# B&R Automation Studio project mappFramework (part 2)

#### HelperMacro.h
```c
/*
* Author: 		B+R
* Contents of this file are modified and extended
*/

/*
 * COPYRIGHT AND PERMISSION NOTICE
 *
 * Copyright (c) 2003 Embedded Unit Project
 *
 * All rights reserved.
 *
 * Permission is hereby granted, free of charge, to any person obtaining
 * a copy of this software and associated documentation files (the
 * "Software"), to deal in the Software without restriction, including
 * without limitation the rights to use, copy, modify, merge, publish,
 * distribute, and/or sell copies of the Software, and to permit persons
 * to whom the Software is furnished to do so, provided that the above
 * copyright notice(s) and this permission notice appear in all copies
 * of the Software and that both the above copyright notice(s) and this
 * permission notice appear in supporting documentation.
 *
 * THE SOFTWARE IS PROVIDED "AS IS", WITHOUT WARRANTY OF ANY KIND,
 * EXPRESS OR IMPLIED, INCLUDING BUT NOT LIMITED TO THE WARRANTIES OF
 * MERCHANTABILITY, FITNESS FOR A PARTICULAR PURPOSE AND NONINFRINGEMENT
 * OF THIRD PARTY RIGHTS. IN NO EVENT SHALL THE COPYRIGHT HOLDER OR
 * HOLDERS INCLUDED IN THIS NOTICE BE LIABLE FOR ANY CLAIM, OR ANY
 * SPECIAL INDIRECT OR CONSEQUENTIAL DAMAGES, OR ANY DAMAGES WHATSOEVER
 * RESULTING FROM LOSS OF USE, DATA OR PROFITS, WHETHER IN AN ACTION OF
 * CONTRACT, NEGLIGENCE OR OTHER TORTIOUS ACTION, ARISING OUT OF OR IN
 * CONNECTION WITH THE USE OR PERFORMANCE OF THIS SOFTWARE.
 *
 * Except as contained in this notice, the name of a copyright holder
 * shall not be used in advertising or otherwise to promote the sale,
 * use or other dealings in this Software without prior written
 * authorization of the copyright holder.
 *
 * $Id: HelperMacro.h,v 1.3 2004/02/10 16:19:29 arms22 Exp $
 */

#ifndef	__HELPERMACRO_H__
#define	__HELPERMACRO_H__

/* Defines the order of test cases */
#define UNITTEST_FIXTURES(fixtures) \
	static const TestFixture	fixtures[] =

/* Standard UnitTest caller without any setup / teardown methods*/
#define UNITTEST_CALLER_TEST(caller,name,fixtures) \
	UNITTEST_CALLER_COMPLETE_EXPLICIT(caller,name,0,0,fixtures,0,0, 0)

/* Standard UnitTest caller with macro setup / teardown for tests*/
#define UNITTEST_CALLER_BASIC(caller,name,fixtures) \
	UNITTEST_CALLER_COMPLETE_EXPLICIT(caller,name,setupTest,teardownTest,fixtures,0,0, 0)

/* UnitTest caller with macro setup / teardown for tests and test set */
#define UNITTEST_CALLER_SET(caller,name,fixtures) \
	UNITTEST_CALLER_COMPLETE_EXPLICIT(caller,name,setupTest,teardownTest,fixtures, setupSet, teardownSet, 0)

/* UnitTest caller with macro setup / teardown for tests and test set and cylic*/
#define UNITTEST_CALLER_COMPLETE(caller,name,fixtures) \
	UNITTEST_CALLER_COMPLETE_EXPLICIT(caller,name,setupTest,teardownTest,fixtures, setupSet, teardownSet, cyclicSetCaller)

/* UnitTest caller with explicit setup / teardown for suite */
#define UNITTEST_CALLER_SET_EXPLICIT(caller,name,sup,tdw,fixtures, setupSuite, teardownSuite) \
	UNITTEST_CALLER_COMPLETE_EXPLICIT(caller,name,sup,tdw,fixtures, setupSuite, teardownSuite, 0)

#ifdef  __cplusplus
/* UnitTest caller with explicit setup / teardown for suite and cylic */
#define UNITTEST_CALLER_COMPLETE_EXPLICIT(caller,name,sup,tdw,fixtures, setupSuite, teardownSuite, cyclicCaller) \
	UNITTEST_TESTSET_DECLARATION caller = new_TestCaller(name,sup,tdw,sizeof(fixtures)/sizeof(fixtures[0]),(TestFixture*)fixtures, setupSuite, teardownSuite, cyclicCaller)

#else

/* UnitTest caller with explicit setup / teardown for suite and cylic */
#define UNITTEST_CALLER_COMPLETE_EXPLICIT(caller,name,sup,tdw,fixtures, setupSuite, teardownSuite, cyclicCaller) \
	 const TestCaller caller = new_TestCaller(name,sup,tdw,sizeof(fixtures)/sizeof(fixtures[0]),(TestFixture*)fixtures, setupSuite, teardownSuite, cyclicCaller)

#endif

#define UNITTEST_CALLER_SKIPPED(caller,name,sup,tdw,fixtures, setupSuite, teardownSuite, cyclicCaller) \
 const TestCaller caller = skipTestCaller(name,sup,tdw,sizeof(fixtures)/sizeof(fixtures[0]),(TestFixture*)fixtures, setupSuite, teardownSuite, cyclicCaller)

/* --------------------------------------*/

/* --------------------------------------*/

typedef struct TestSetActive
{
	BOOL			active;
	TestCallerRef 	set;
} TestSetActive;

typedef struct TestSetList
{
	UINT 			nrOfTestSets;
	UINT 			currentTestSet;
	TestSetActive 	*list;
} TestSetList;

/* Defines the order of test sets.
Should look like this
UNITTEST_TESTSET_FIXTURES(fixtures)
{
	new_TestSet(testSet_1),
	new_TestSet(testSet_2),
	new_TestSet(testSet_3)
}*/
#define UNITTEST_TESTSET_FIXTURES(fixtures) \
	static TestSetActive	fixtures[] =

/* Adds a test set with description to the fixture of test sets.
See UNITTEST_TESTSET_FIXTURES() */
#define new_TestSet(testcaller)\
	{\
		1,\
		(TestCallerRef)&testcaller,\
	}

/* Adds a test set with description to the fixture of test sets.
See UNITTEST_TESTSET_FIXTURES() */
#define skipTestSet(testcaller)\
	{\
		1,\
		(TestCallerRef)&testcaller,\
	}

/* Adds a test set with description to the fixture of test sets.
See UNITTEST_TESTSET_FIXTURES() */
#define disabledTestSet(testcaller)\
	{\
		0,\
		(TestCallerRef)&testcaller,\
	}

/* Defines the test set list handling structure*/
#define UNTITTEST_TESTSET_HANDLER() \
TestSetList setList = {\
	sizeof(utTestSets) / sizeof(TestSetActive), \
	0, \
	(TestSetActive*)&utTestSets\
	}

#endif/*__HELPERMACRO_H__*/
```

#### utRunner.h
```c
/********************************************************************
 * COPYRIGHT B+R
 ********************************************************************
 * Library: utRunner
 * File: utRunner.h
 * Author: B+R
 *******************************************************************/

#ifndef	__UT_RUNNER_H__
#define	__UT_RUNNER_H__

#include <bur/plctypes.h>

#include "UnitTest.h"
#include "UtMgr.h"
#include "include/TestCaller.h"

#ifdef __cplusplus
extern "C"
{
#endif

void utInit(UtMgrTestSuite_typ *TestSuiteRef);
void utCyclic(UtMgrTestSuite_typ *TestSuiteRef);
void utExit(UtMgrTestSuite_typ *TestSuiteRef);

#ifdef __cplusplus
};
#endif

#endif/*__UT_RUNNER_H__*/
```

#### Test.h
```c
/*
* Author: 		B+R
* Contents of this file are modified and extended
*/

/*
 * COPYRIGHT AND PERMISSION NOTICE
 *
 * Copyright (c) 2003 Embedded Unit Project
 *
 * All rights reserved.
 *
 * Permission is hereby granted, free of charge, to any person obtaining
 * a copy of this software and associated documentation files (the
 * "Software"), to deal in the Software without restriction, including
 * without limitation the rights to use, copy, modify, merge, publish,
 * distribute, and/or sell copies of the Software, and to permit persons
 * to whom the Software is furnished to do so, provided that the above
 * copyright notice(s) and this permission notice appear in all copies
 * of the Software and that both the above copyright notice(s) and this
 * permission notice appear in supporting documentation.
 *
 * THE SOFTWARE IS PROVIDED "AS IS", WITHOUT WARRANTY OF ANY KIND,
 * EXPRESS OR IMPLIED, INCLUDING BUT NOT LIMITED TO THE WARRANTIES OF
 * MERCHANTABILITY, FITNESS FOR A PARTICULAR PURPOSE AND NONINFRINGEMENT
 * OF THIRD PARTY RIGHTS. IN NO EVENT SHALL THE COPYRIGHT HOLDER OR
 * HOLDERS INCLUDED IN THIS NOTICE BE LIABLE FOR ANY CLAIM, OR ANY
 * SPECIAL INDIRECT OR CONSEQUENTIAL DAMAGES, OR ANY DAMAGES WHATSOEVER
 * RESULTING FROM LOSS OF USE, DATA OR PROFITS, WHETHER IN AN ACTION OF
 * CONTRACT, NEGLIGENCE OR OTHER TORTIOUS ACTION, ARISING OUT OF OR IN
 * CONNECTION WITH THE USE OR PERFORMANCE OF THIS SOFTWARE.
 *
 * Except as contained in this notice, the name of a copyright holder
 * shall not be used in advertising or otherwise to promote the sale,
 * use or other dealings in this Software without prior written
 * authorization of the copyright holder.
 *
 * $Id: Test.h,v 1.4 2004/02/10 16:19:29 arms22 Exp $
 */
#ifndef	__TEST_H__
#define	__TEST_H__

typedef struct __TestResult		TestResult;
typedef struct __TestResult	*TestResultRef;/*downward compatible*/

typedef struct __TestImplement	TestImplement;
typedef struct __TestImplement	*TestImplementRef;/*downward compatible*/

typedef enum testStatusEnum
{
    ut_BUSY = 0,
    ut_DONE = 1,
    ut_ABORT = 2
} testStatusEnum;

typedef char* 			(*TestNameFunction)(void *);

typedef testStatusEnum	(*TestRunFunction)(void *, TestResult *);
typedef int				(*TestCountTestCasesFunction)(void *);

typedef enum testStateEnum
{
    stateStart, 	/* print something */
    stateSetup,
    stateRun,
    stateTearDown,
    stateEnd,		/* print something */
    stateDefault, 	/* last state*/
} testStateEnum;

struct __TestImplement
{
	TestNameFunction 			name;
	TestRunFunction 			run;
	TestCountTestCasesFunction countTestCases;
};

typedef struct __Test	Test;
typedef struct __Test	*TestRef;/*downward compatible*/

struct __Test
{
	TestImplement *isa;
};

#define Test_name(s)			((Test*)s)->isa->name(s)
#define Test_run(s,r)			((Test*)s)->isa->run(s,r)
#define Test_countTestCases(s)	((Test*)s)->isa->countTestCases(s)

#endif/*__TEST_H__*/
```

#### TestListener.h
```c
/*
* Author: 		B+R
* Contents of this file are modified and extended
*/

/*
 * COPYRIGHT AND PERMISSION NOTICE
 *
 * Copyright (c) 2003 Embedded Unit Project
 *
 * All rights reserved.
 *
 * Permission is hereby granted, free of charge, to any person obtaining
 * a copy of this software and associated documentation files (the
 * "Software"), to deal in the Software without restriction, including
 * without limitation the rights to use, copy, modify, merge, publish,
 * distribute, and/or sell copies of the Software, and to permit persons
 * to whom the Software is furnished to do so, provided that the above
 * copyright notice(s) and this permission notice appear in all copies
 * of the Software and that both the above copyright notice(s) and this
 * permission notice appear in supporting documentation.
 *
 * THE SOFTWARE IS PROVIDED "AS IS", WITHOUT WARRANTY OF ANY KIND,
 * EXPRESS OR IMPLIED, INCLUDING BUT NOT LIMITED TO THE WARRANTIES OF
 * MERCHANTABILITY, FITNESS FOR A PARTICULAR PURPOSE AND NONINFRINGEMENT
 * OF THIRD PARTY RIGHTS. IN NO EVENT SHALL THE COPYRIGHT HOLDER OR
 * HOLDERS INCLUDED IN THIS NOTICE BE LIABLE FOR ANY CLAIM, OR ANY
 * SPECIAL INDIRECT OR CONSEQUENTIAL DAMAGES, OR ANY DAMAGES WHATSOEVER
 * RESULTING FROM LOSS OF USE, DATA OR PROFITS, WHETHER IN AN ACTION OF
 * CONTRACT, NEGLIGENCE OR OTHER TORTIOUS ACTION, ARISING OUT OF OR IN
 * CONNECTION WITH THE USE OR PERFORMANCE OF THIS SOFTWARE.
 *
 * Except as contained in this notice, the name of a copyright holder
 * shall not be used in advertising or otherwise to promote the sale,
 * use or other dealings in this Software without prior written
 * authorization of the copyright holder.
 *
 * $Id: TestListener.h,v 1.4 2004/02/10 16:19:29 arms22 Exp $
 */
#ifndef	__TESTLISTENER_H__
#define	__TESTLISTENER_H__

typedef struct __TestListnerImplement	TestListnerImplement;
typedef struct __TestListnerImplement	*TestListnerImplementRef;/*downward compatible*/

typedef void(*TestListnerStartTestCallBack)(void *,void *);
typedef void(*TestListnerEndTestCallBack)(void *,void *);
typedef void(*TestListnerSkippedTestCallBack)(void *,void *);

typedef void(*TestListnerAddFailureCallBack)(void *,void *,const char *,unsigned long,const char *);

typedef void(*TestListnerAddPassedCallBack)(void *,void *,const char *,unsigned long,const char *);
typedef void(*TestListnerAddInfoCallBack)(void *,void *,const char *,unsigned long,const char *);
typedef void(*TestListnerAddAbortCallBack)(void *,void *,const char *,unsigned long,const char *);
typedef void(*TestListnerLogCallBack)(void *,void *,const char *,unsigned long,const char *, signed short);

struct __TestListnerImplement
{
	TestListnerStartTestCallBack 	startTest;
	TestListnerEndTestCallBack 		endTest;
	TestListnerSkippedTestCallBack 	skippedTest;
	TestListnerAddFailureCallBack 	addFailure;
	TestListnerAddPassedCallBack 	addPassed;
	TestListnerAddInfoCallBack 		addInfo;
	TestListnerAddAbortCallBack 	addAbort;
	TestListnerLogCallBack			doLog;
};

/*typedef struct __TestListner	TestListner;*/	/*->TestResult.h*/
/*typedef struct __TestListner*	TestListnerRef;*/	/*->TestResult.h*/

struct __TestListner
{
	TestListnerImplement *isa;
};

#define TestListner_startTest(s,t)			((TestListner*)s)->isa->startTest(s,t)
#define TestListner_endTest(s,t)			((TestListner*)s)->isa->endTest(s,t)
#define TestListner_skippedTest(s,t)			((TestListner*)s)->isa->skippedTest(s,t)

#define TestListner_addFailure(s,t,m,l,f)	((TestListner*)s)->isa->addFailure(s,t,m,l,f)
#define TestListner_addPassed(s,t,m,l,f)	((TestListner*)s)->isa->addPassed(s,t,m,l,f)
#define TestListner_addInfo(s,t,m,l,f)		((TestListner*)s)->isa->addInfo(s,t,m,l,f)
#define TestListner_addAbort(s,t,m,l,f)		((TestListner*)s)->isa->addAbort(s,t,m,l,f)
#define TestListener_doLog(s,t,m,l,f,e)		if(s)(((TestListner*)s)->isa->doLog(s,t,m,l,f,e))
#endif/*__TESTLISTENER_H__*/
```

#### TestResult.h
```c
/*
* Author: 		B+R
* Contents of this file are modified and extended
*/

/*
* COPYRIGHT AND PERMISSION NOTICE
*
* Copyright (c) 2003 Embedded Unit Project
*
* All rights reserved.
*
* Permission is hereby granted, free of charge, to any person obtaining
* a copy of this software and associated documentation files (the
* "Software"), to deal in the Software without restriction, including
* without limitation the rights to use, copy, modify, merge, publish,
* distribute, and/or sell copies of the Software, and to permit persons
* to whom the Software is furnished to do so, provided that the above
* copyright notice(s) and this permission notice appear in all copies
* of the Software and that both the above copyright notice(s) and this
* permission notice appear in supporting documentation.
*
* THE SOFTWARE IS PROVIDED "AS IS", WITHOUT WARRANTY OF ANY KIND,
* EXPRESS OR IMPLIED, INCLUDING BUT NOT LIMITED TO THE WARRANTIES OF
* MERCHANTABILITY, FITNESS FOR A PARTICULAR PURPOSE AND NONINFRINGEMENT
* OF THIRD PARTY RIGHTS. IN NO EVENT SHALL THE COPYRIGHT HOLDER OR
* HOLDERS INCLUDED IN THIS NOTICE BE LIABLE FOR ANY CLAIM, OR ANY
* SPECIAL INDIRECT OR CONSEQUENTIAL DAMAGES, OR ANY DAMAGES WHATSOEVER
* RESULTING FROM LOSS OF USE, DATA OR PROFITS, WHETHER IN AN ACTION OF
* CONTRACT, NEGLIGENCE OR OTHER TORTIOUS ACTION, ARISING OUT OF OR IN
* CONNECTION WITH THE USE OR PERFORMANCE OF THIS SOFTWARE.
*
* Except as contained in this notice, the name of a copyright holder
* shall not be used in advertising or otherwise to promote the sale,
* use or other dealings in this Software without prior written
* authorization of the copyright holder.
*
* $Id: TestResult.h,v 1.7 2004/02/10 16:19:29 arms22 Exp $
*/
#ifndef	__TESTRESULT_H__
#define	__TESTRESULT_H__

#ifdef	__cplusplus
extern "C" {
#endif

/*typedef struct __TestResult		TestResult;*//* -> Test.h*/
/*typedef struct __TestResult*		TestResultRef;*//* -> Test.h*/

typedef struct __TestListner	TestListner;
typedef struct __TestListner	*TestListnerRef;/*downward compatible*/

struct __TestResult
{
	unsigned short runCount;
	unsigned short failureCount;
	unsigned short passedCount;
	unsigned short infoCount;
	unsigned short summarizedCount;
	unsigned short abortCount;
	unsigned short skippedTestCount;
	unsigned short suceessedTestCount;
	TestListner *listener;
};

#define new_TestResult(listener)\
{\
	0,\
	0,\
	0,\
	0,\
	0,\
	0,\
	0,\
	0,\
	(TestListner*)listener\
}

void TestResult_init(TestResult *self,TestListner *listner);
void TestResult_startTest(TestResult *self,Test *test);
void TestResult_endTest(TestResult *self,Test *test);
void TestResult_skipTest(TestResult *self,Test *test);

void TestResult_addFailure(TestResult *self,Test *test,const char *msg,unsigned long line,const char *file);
void TestResult_addPassed(TestResult *self,Test *test,const char *msg,unsigned long line,const char *file);
void TestResult_addInfo(TestResult *self,Test *test,const char *msg,unsigned long line,const char *file);
void TestResult_addAbort(TestResult *self,Test *test,const char *msg,unsigned long line,const char *file);

#ifdef	__cplusplus
}
#endif

#endif/*__TESTRESULT_H__*/
```

### Package Logical/Infrastructure/TS_UnitTest/Samples/Tests_Program - Unit test sample

### Library Logical/Infrastructure/TS_UnitTest/Samples/Tests_Program/SPLMyCalc (IEC)
Depends on: Runtime

#### SPLMyCalc.st
```iecst
(********************************************************************
 * COPYRIGHT -- Bernecker + Rainer
 ********************************************************************
 * Library: SPLMyCalc
 * File: SPLMyCalc.st
 * Author: B+R
 ********************************************************************
 * Implementation of library SPLMyCalc
 *******************************************************************

// This can be used as a sample for  Test Driven Development (TDD)/ Test First Development
Steps (in a nutshell):
    o Define your API (FB, functions, ...)
		 this is already done for the FB MyCalc
	o Create a new test program (by using the template)
	o Write a test case (e.g. Addition) for this FB.
		The tests should describe the expected behavior.
	o Transfer the test program to the target and run the test in the test view
		The test case will fail
	o Implement this FB (Addition), build and transfer, then run the test again
		The test case will pass
	o Write next test (e.g. Subtraction).
	..
	o Write test for MIN / MAX (underflow/overflow)
   	o Run the tests to verify your implementation.

Note:
	The sample test program in SPL_MyCalcLib_C provides some test cases using this FB.

FUNCTION_BLOCK MyCalculator

	Status := ERR_NOTIMPLEMENTED;

END_FUNCTION_BLOCK
```

### Program Logical/Infrastructure/TS_UnitTest/Samples/Tests_Program/Tests_MyCalcLib_C/SPL_CalcTest (ANSIC) - Tests SPLMyCalc with library "UnitTest"

#### testSuite.c - Handling of program and test suite
```c
/********************************************************************
 * COPYRIGHT -- Bernecker + Rainer
 ********************************************************************
 * Program: SPL_CalcTest
 * Author: B+R
 ********************************************************************
 * Test registration and handshake
 ********************************************************************/

#include <bur/plctypes.h>

#ifdef _DEFAULT_INCLUDES
#include <AsDefault.h>
#endif

#include "UnitTest.h"

void _INIT initTestSuite(void)
{
	utInit(&Testsuite);
}

void _CYCLIC cyclicWithTest(void)
{
	utCyclic(&Testsuite);
}

void _EXIT exitTestSuite(void)
{
	utExit(&Testsuite);
}
```

#### testSet_MyCalcLib_Addition.c - Groups test cases for addition
```c
/********************************************************************
 * COPYRIGHT -- Bernecker + Rainer
 ********************************************************************
 * Program: SPL_CalcTest
 * Author: B+R
 ********************************************************************
 * Test set implementation
 ********************************************************************/

#include <bur/plctypes.h>

#ifdef _DEFAULT_INCLUDES
#include <AsDefault.h>
#endif

#include "UnitTest.h"

_TEST test_Add(void)
{
	/* initialize functionblock parameters */
	instMyCalc.CalcOperator = splMyCalcOPERATOR_ADD;
	instMyCalc.Param1   = 1;
	instMyCalc.Param2   = 2;
	/* call synchron functionblock */
	MyCalculator(&instMyCalc);

	/* check result */
	TEST_ASSERT_EQUAL_INT(3, instMyCalc.Result);
	TEST_ASSERT_EQUAL_INT(ERR_OK, instMyCalc.Status);

	/* test is done */
	TEST_DONE;
}

_TEST testResetOutputParam(void)
{

	/* Do any calculation with a result != 0  */
	instMyCalc.CalcOperator = splMyCalcOPERATOR_ADD;
	instMyCalc.Param1   = 1;
	instMyCalc.Param2   = 2;
	/* call synchron functionblock */
	MyCalculator(&instMyCalc);
	/* Please note: the result of the calculation isn't checked as this is not subject of this test case.	 */

	instMyCalc.CalcOperator = splMyCalcOPERATOR_RESET_OUTPUTS;
	/* call synchron functionblock */
	MyCalculator(&instMyCalc);

	/* check result */
	TEST_ASSERT_EQUAL_INT(0, instMyCalc.Result);
	TEST_ASSERT_EQUAL_INT(ERR_OK, instMyCalc.Status);

	/* test is done */
	TEST_DONE;

}

/* This test case shows an example of a test case that can be "false positive".
	As long as MyCalculator() is not implemented, this test passes.
	As long as instMyCalc.Result already is 0 when this test case will be called, it doesn't check wether the FB was called at all.
	--> There are several methods, to verify the FB was called and changed the variables that are used to prove functionality:
	Choose other parameter for an addition with negative values
	Before calling the FB set the output to any other value than the expected result. (e.g. By using _SETUP_TEST() and / or _TEARDOWN_TEST() )
	...

*/
_TEST test_Addition_negValue_badExampleParameter(void)
{
	/* initialize functionblock parameters */
	instMyCalc.CalcOperator = splMyCalcOPERATOR_ADD;
	instMyCalc.Param1   = -1;
	instMyCalc.Param2   = 1;
	/* call synchron functionblock */
	MyCalculator(&instMyCalc);

	/* check result */
	TEST_ASSERT_EQUAL_INT(0, instMyCalc.Result);
	TEST_ASSERT_EQUAL_INT(ERR_OK, instMyCalc.Status);

	/* test is done */
	TEST_DONE;
}

_TEST test_Addition_negValue(void)
{
	/* initialize functionblock parameters */
	instMyCalc.CalcOperator = splMyCalcOPERATOR_ADD;
	instMyCalc.Param1   = -1;
	instMyCalc.Param2   = 3;
	/* call synchron functionblock */
	MyCalculator(&instMyCalc);

	/* check result */
	TEST_ASSERT_EQUAL_INT(2, instMyCalc.Result);
	TEST_ASSERT_EQUAL_INT(ERR_OK, instMyCalc.Status);

	/* test is done */
	TEST_DONE;
}

/*
B+R UnitTest: This is generated code.
Do not edit! Do not move!
Description: UnitTest Testprogramm infrastructure (TestSet).
LastUpdated: 2015-04-14 12:04:18Z
By B+R UnitTest Helper Version: 2.0.0.0
*/
UNITTEST_FIXTURES(fixtures)
{
	new_TestFixture("test_Add", test_Add),
	new_TestFixture("testResetOutputParam", testResetOutputParam),
	new_TestFixture("test_Addition_negValue_badExampleParameter", test_Addition_negValue_badExampleParameter),
	new_TestFixture("test_Addition_negValue", test_Addition_negValue),
};

UNITTEST_CALLER_COMPLETE_EXPLICIT(testSet_MyCalcLib_Addition, "testSet_MyCalcLib_Addition", 0, 0, fixtures, 0, 0, 0);
```

#### testSet_MyCalcLib_Mult_Div.c - Groups test cases for multiplication and division
```c
/********************************************************************
 * COPYRIGHT -- Bernecker + Rainer
 ********************************************************************
 * Program: SPL_CalcTest
 * Author: B+R
 ********************************************************************
 * Test set implementation
 ********************************************************************/

#include <bur/plctypes.h>

#ifdef _DEFAULT_INCLUDES
#include <AsDefault.h>
#endif

#include "UnitTest.h"

_TEST test_Multiplication(void)
{
	/* initialize functionblock parameters */
	instMyCalc.CalcOperator = splMyCalcOPERATOR_MULTIPLICATION;
	instMyCalc.Param1   = 4;
	instMyCalc.Param2   = 4;
	/* call synchron functionblock */
	MyCalculator(&instMyCalc);
	/* check result */
	TEST_ASSERT_EQUAL_INT(16, instMyCalc.Result);
	TEST_ASSERT_EQUAL_INT(ERR_OK, instMyCalc.Status);
	/* test is done */
	TEST_DONE;
}

_TEST test_Division(void)
{
	/* initialize functionblock parameters */
	instMyCalc.CalcOperator = splMyCalcOPERATOR_DIVISION;
	instMyCalc.Param1   = 4;
	instMyCalc.Param2   = 4;
	/* call synchron functionblock */
	MyCalculator(&instMyCalc);

	/* check result */
	TEST_ASSERT_EQUAL_INT(1, instMyCalc.Result);
	TEST_ASSERT_EQUAL_INT(ERR_OK, instMyCalc.Status);

	/* test is done */
	TEST_DONE;
}

/*
B+R UnitTest: This is generated code.
Do not edit! Do not move!
Description: UnitTest Testprogramm infrastructure (TestSet).
LastUpdated: 2015-04-14 12:04:18Z
By B+R UnitTest Helper Version: 2.0.0.0
*/
UNITTEST_FIXTURES(fixtures)
{
	new_TestFixture("test_Multiplication", test_Multiplication),
	new_TestFixture("test_Division", test_Division),
};

UNITTEST_CALLER_COMPLETE_EXPLICIT(testSet_MyCalcLib_Mult_Div, "testSet_MyCalcLib_Mult_Div", 0, 0, fixtures, 0, 0, 0);
```

### Program Logical/Infrastructure/TS_UnitTest/Samples/Tests_Program/Tests_MyCalcLib_C/SPL_CalcTest_Variants (ANSIC) - Examples how to avoid duplicated test code (advanced)

#### variables.var - PVs for the program and test suite
```iecst
(********************************************************************
 * COPYRIGHT -- Bernecker + Rainer
 ********************************************************************
 * Program: SPL_CalcTest_Variants
 * Author: B+R
 ********************************************************************
 * Local variables of program SPL_CalcTest_Variants
 * General variables - do not change
 ********************************************************************)
(*Describe the test*)
VAR
	Testsuite : UtMgrTestSuite := (Name:='SPL_CalcTest_Variants',Description:='Tests for MyCalc',Type:=utMgrTEST_TYPE_C,MetaInformation:='Some Meta Information can be added here');
END_VAR
(*Variables used in the tests*)
VAR
	instMyCalc : MyCalculator := (0);
END_VAR
```

### Package Logical/Infrastructure/TS_UnitTest/Samples/Framework_Extension_With_Custom_Asserts - Custom asserts

### Library Logical/Infrastructure/TS_UnitTest/Samples/Framework_Extension_With_Custom_Asserts/LibAssert1 (ANSIC) - Sample library: Creation of custom asserts

#### LibAssert1_REAL_ArrayAsserts.h
```c
/********************************************************************
 * COPYRIGHT -- Bernecker + Rainer
 ********************************************************************
 * Library: LibAssert1
 * File: LibAssert1_REAL_ArrayAsserts.h
 * Author: B+R
 *******************************************************************/

#include <bur/plctypes.h>
#include "UnitTest.h"

#ifdef __cplusplus
extern "C"
{
#endif

	/* Dummies for smart edit autocompletion.
	See below for the real macros used by the compiler  */
#ifdef _SMART_EDIT_DUMMY_

	/* This assert checks two arrays of floats for equality. TEST_FLOAT_PRECISION is used as default Delta.

	Note: An assert like this is generally more readable and meaningful than multiple TEST_ASSERT_EQUAL_FLOAT().
	It informs about how many entries failed in total and shows the first NR_OF_DETAILED_ENTRIES_TO_SHOW together with the array index the failure occured. */
	BOOL SPL_ASSERT_ARRAY_EQUAL_REAL(REAL *expected[], REAL *actual[], UDINT nrOfEntries);

	/* This assert checks two arrays of floats for equality with an accepted delta per entry

	Note: An assert like this is generally more readable and meaningful than multiple TEST_ASSERT_FLOAT_WITHIN().
	It informs about how many entries failed in total and shows the first NR_OF_DETAILED_ENTRIES_TO_SHOW together with the array index the failure occured.
	*/
	BOOL SPL_ASSERT_ARRAY_REAL_WITHIN(REAL *delta[], REAL *expected[], REAL *actual[], UDINT nrOfEntries);

#endif

	/*------------------------------------------------------------*/

	/* Prototyping of functions.
	These declaration of functions are used by the compiler to check number and type of arguments. */
	BOOL spl_assertImplRealArrayEqual(const REAL delta,
	                                  const REAL *expected,
	                                  const REAL *actual,
	                                  const unsigned long nrOfEntries,
	                                  unsigned long line, const char *file);

	BOOL spl_assertImplRealArrayWithin(const REAL *delta,
	                                   const REAL *expected,
	                                   const REAL *actual,
	                                   const unsigned long nrOfEntries,
	                                   unsigned long line, const char *file);

	/* Makros used in the test implementation.
	The macro passes the location information to the implemented assert. */

#define SPL_ASSERT_ARRAY_EQUAL_REAL(expected, actual, nrOfEntries)	\
	spl_assertImplRealArrayEqual((REAL)TEST_FLOAT_PRECISION, expected, actual, nrOfEntries, (unsigned long) __LINE__, __FILE__)

#define SPL_ASSERT_ARRAY_REAL_WITHIN(delta, expected, actual, nrOfEntries)	\
	spl_assertImplRealArrayWithin(delta, expected, actual, nrOfEntries,  (unsigned long) __LINE__, __FILE__)

#ifdef __cplusplus
};
#endif
```

#### LibAssert1_ThresholdAssert.h
```c
/********************************************************************
 * COPYRIGHT -- Bernecker + Rainer
 ********************************************************************
 * Library: LibAssert1
 * File: LibAssert1_ThresholdAssert.h
 * Author: B+R
 *******************************************************************/

#include <bur/plctypes.h>

#include <bur/plctypes.h>
#include "UnitTest.h"

#ifdef __cplusplus
extern "C"
{
#endif

/* Dummies for smart edit autocompletion.
See below for the real macros used by the compiler  */
#ifdef _SMART_EDIT_DUMMY_
	/* This asserts checks (actual < threshold) */
	BOOL SPL_ASSERT_UPPER_BOUNDARY(DINT threshold, DINT actual);
#endif

/*------------------------------------------------------------*/

/* Prototyping of functions.
These declaration of functions are used by the compiler to check number and type of arguments. */
BOOL spl_assertUpperBoundary_DINT(const DINT threshold, const DINT actual, unsigned long line, const char *file);

/* Macros used in the test implementation.
The macro passes the location information to the implemented assert. */
#define SPL_ASSERT_UPPER_BOUNDARY(threshold, actual) 	\
	spl_assertUpperBoundary_DINT(threshold, actual, (unsigned long) __LINE__, __FILE__)

#ifdef __cplusplus
};
#endif
```

#### LibAssert1_REAL_ArrayAsserts.c
```c
/********************************************************************
 * COPYRIGHT -- Bernecker + Rainer
 ********************************************************************
 * Library: LibAssert1
 * File: LibAssert1_REAL_ArrayAsserts.c
 * Author: B+R
 *******************************************************************/

#include <bur/plctypes.h>

#include "asbrstr.h"
#include "LibAssert1_REAL_ArrayAsserts.h"

#define TRUE 1
#define FALSE 0

#define NR_OF_DETAILED_ENTRIES_TO_SHOW 10

/* Tests each REAL in the array for equality in range
Returns true if passed, false otherwise
delta: allowed tolerance (floats are not exact values)
expected: array of expected REAL values
acutal: array of REAL values under test
nrOfEntries: number of entries in array
line: location information
file: location information
*/
BOOL spl_assertImplRealArrayWithin(const REAL *delta,
                                   const REAL *expected, 	const REAL *actual, const unsigned long nrOfEntries,
                                   unsigned long line, const char *file)
{
	unsigned long i = 0;
	unsigned long countFail = 0;
	STRING buffer[100];
	STRING numbuf[30];

	/*------------------------------------------------------------*/
	for(i = 0; i < nrOfEntries; i++)
	{
		REAL diff = actual[i] - expected[i];
		REAL pos_delta = delta[i];

		if (diff < 0)
		{
			/* use absolute (positive) value */
			diff = 0.0f - diff;
		}
		if (pos_delta < 0)
		{
			/* use absolute (positive) value */
			pos_delta = 0.0f - pos_delta;
		}

		/* Check */
		if (pos_delta < diff)
		{
			/* count the failures */
			countFail++;

			/* for the first NR_OF_DETAILED_ENTRIES_TO_SHOW failures generate an informational message) */
			if(countFail < NR_OF_DETAILED_ENTRIES_TO_SHOW)
			{
				brsstrcpy((unsigned long) buffer, (unsigned long) "At array index ");
				brsitoa((int)i, (unsigned long)numbuf);
				brsstrcat((unsigned long) buffer, (unsigned long) numbuf);

				brsstrcat((unsigned long) buffer, (unsigned long) ": exp ");
				brsftoa((REAL)expected[i], (unsigned long)numbuf);
				brsstrcat((unsigned long) buffer, (unsigned long) numbuf);

				brsstrcat((unsigned long) buffer, (unsigned long)" was ");
				brsftoa((REAL)actual[i], (unsigned long)numbuf);
				brsstrcat((unsigned long) buffer, (unsigned long) numbuf);

				addInfo(buffer, line, file);
			}
		}
	}/* end for */
	/*------------------------------------------------------------*/
	/* All entries checked, generate notification for test report */
	if(0 == countFail)
	{
		addPassed("", line, file);
		return TRUE;
	}
	else
	{
		brsitoa(countFail, (unsigned long)numbuf);
		brsstrcpy((unsigned long)buffer, (unsigned long)numbuf);
		brsstrcat((unsigned long)buffer, (unsigned long)" failures occured in array ");
		addFailure(buffer, line, file);
		return FALSE;
	}
}

/* Tests each REAL in the array for equality
Returns true if passed, false otherwise
delta: allowed tolerance (floats are not exact values)
expected: array of expected REAL values
acutal: array of REAL values under test
nrOfEntries: number of entries in array
line: location information
file: location information
*/
BOOL spl_assertImplRealArrayEqual(const REAL delta,
                                  const REAL *expected, 	const REAL *actual, const unsigned long nrOfEntries,
                                  unsigned long line, const char *file)
{
	unsigned long i = 0;
	char countFail = 0;
	STRING buffer[100];
	STRING numbuf[30];

	/*------------------------------------------------------------*/
	for(i = 0; i < nrOfEntries; i++)
	{
		REAL diff = actual[i] - expected[i];
		REAL pos_delta = delta * (REAL)(expected[i]);

		if (diff < 0)
		{
			/* use absolute (positive) value */
			diff = 0.0f - diff;
		}
		if (pos_delta < 0)
		{
			/* use absolute (positive) value */
			pos_delta = 0.0f - pos_delta;
		}

		/* Check */
		if (pos_delta < diff)
		{
			/* count the failures */
			countFail++;

			/* for the first NR_OF_DETAILED_ENTRIES_TO_SHOW failures generate an informational message) */
			if(countFail < NR_OF_DETAILED_ENTRIES_TO_SHOW)
			{
				brsstrcpy((unsigned long) buffer, (unsigned long) "At array index ");
				brsitoa((int)i, (unsigned long) numbuf);
				brsstrcat((unsigned long) buffer, (unsigned long) numbuf);

				brsstrcat((unsigned long) buffer, (unsigned long) ": exp ");
				brsftoa((REAL)expected[i], (unsigned long)numbuf);
				brsstrcat((unsigned long) buffer, (unsigned long) numbuf);

				brsstrcat((unsigned long) buffer, (unsigned long) " was ");
				brsftoa((REAL)actual[i], (unsigned long)numbuf);
				brsstrcat((unsigned long) buffer, (unsigned long) numbuf);

				addInfo(buffer, 0, 0);
			}
		}
	}/* end for */

	/*------------------------------------------------------------*/
	/* All entries checked, generate notification for test report */
	if(0 == countFail)
	{
		addPassed("", line, file);
		return TRUE;
	}
	else
	{
		brsitoa(countFail, (unsigned long)numbuf);
		brsstrcpy((unsigned long)buffer, (unsigned long)numbuf);
		brsstrcat((unsigned long)buffer,(unsigned long) " failures occured in array ");
		addFailure(buffer, line, file);
		return FALSE;
	}
}
```

### Program Logical/Infrastructure/TS_UnitTest/Samples/Framework_Extension_With_Custom_Asserts/SPL_AssertsEx (ANSIC) - This sample uses custom asserts defined in LibAssert1

#### README.txt
```
Please note

The samples in this program provides no good programming style!
They are solely for demonstrating the behavior of the framework.
Bad style:
	o	There is no test of any function or FB, just asserts failing or passing (depending on PV values)
	o	Expectations are variables and no constants
	o	Results are constants instead of results / outputs
	o	Mulitple asserts per Test Case
```

#### testSuite.var
```iecst
(********************************************************************
 * COPYRIGHT -- Bernecker + Rainer
 ********************************************************************
 * Program: SPL_AssertsEx
 * Author: B+R
 ********************************************************************
 * Local variables of program SPL_AssertsEx
 * General variables
 ********************************************************************)
VAR
	Testsuite : UtMgrTestSuite := (Name:='SPL_CustomAsserts',Description:='The sample custom asserts are defined in LibAssert1. This test shows their usage.',Type:=utMgrTEST_TYPE_C);
END_VAR
```

#### autoGeneratedFile.c
```c
/*
B+R UnitTest: This is generated code.
Do not edit! Do not move!
Description: UnitTest Testprogramm infrastructure (List of TestSets).
LastUpdated: 2015-04-14 12:04:08Z
By B+R UnitTest Helper Version: 2.0.0.0
*/
#include "UnitTest.h"

UNITTEST_TESTSET_DECLARATION  testSet_AssertsExt;

UNITTEST_TESTSET_FIXTURES(utTestSets)
{
	new_TestSet(testSet_AssertsExt),
};
UNTITTEST_TESTSET_HANDLER();
```

### Package Logical/Infrastructure/TS_UnitTest/Samples/Framework_Features - Framework features

### Program Logical/Infrastructure/TS_UnitTest/Samples/Framework_Features/SPL_Asserts (ANSIC) - Available basic asserts

#### varAsserts.var
```iecst
(********************************************************************
 * COPYRIGHT -- Bernecker + Rainer
 ********************************************************************
 * Program: SPL_Asserts
 * Author: B+R
 ********************************************************************
 * Local variables of program SPL_Asserts
 * For test set testSet_Asserts.c
 ********************************************************************)
VAR
	Buffer1 : ARRAY[0..9] OF USINT := [10(0)];
	Buffer2 : ARRAY[0..19] OF USINT := [20(0)];
	MySecondVar : UDINT := 2;
	Pointer : REFERENCE TO UDINT;
	ConditionFlag : BOOL := FALSE;
END_VAR
(*Strings*)
VAR
	String1 : STRING[80] := '';
	String2 : STRING[80] := '';
	WString1 : WSTRING[80] := "World";
	WString2 : WSTRING[80] := "Hello";
END_VAR
(*Integer*)
VAR
	Si1 : SINT := 0;
	Si2 : SINT := 0;
	Usi1 : USINT := 0;
	Usi2 : USINT := 0;
	I1 : INT := 0;
	I2 : INT := 0;
	Ui1 : UINT := 0;
	Ui2 : UINT := 0;
	Di1 : DINT := 0;
	Di2 : DINT := 0;
	Udi1 : UDINT := 0;
	Udi2 : UDINT := 0;
END_VAR
(*Floatingpoint*)
VAR
	LReal2 : REAL;
	LRealDeltaForComparison : REAL;
	LReal1 : REAL;
	Real2 : REAL;
	RealDeltaForComparison : REAL;
	Real1 : REAL;
END_VAR
```

#### autoGeneratedFile.c
```c
/*
B+R UnitTest: This is generated code.
Do not edit! Do not move!
Description: UnitTest Testprogramm infrastructure (List of TestSets).
LastUpdated: 2015-04-14 12:03:48Z
By B+R UnitTest Helper Version: 2.0.0.0
*/
#include "UnitTest.h"

UNITTEST_TESTSET_DECLARATION  testSet_Asserts;

UNITTEST_TESTSET_FIXTURES(utTestSets)
{
	new_TestSet(testSet_Asserts),
};
UNTITTEST_TESTSET_HANDLER();
```

#### testSet_Asserts.c
```c
/********************************************************************
* COPYRIGHT -- Bernecker + Rainer
********************************************************************
* Program: SPL_Asserts
* Author: B+R
********************************************************************
* This test set shows the available asserts of the UnitTest library
********************************************************************/

#include <bur/plctypes.h>

#ifdef _DEFAULT_INCLUDES
#include <AsDefault.h>
#endif

#include "UnitTest.h"

/* Executed before each test case */
_SETUP_TEST(void)
{
	MySecondVar = 2;

	TEST_DONE;
}

/* Executed after each test case */
_TEARDOWN_TEST(void)
{
	TEST_DONE;
}

_TEST test_int(void)
{
	TEST_ASSERT_EQUAL_INT(	Usi1, 	Usi2);
	TEST_ASSERT_EQUAL_INT( 	Si1,	Si2 );
	TEST_ASSERT_EQUAL_INT( 	Ui1, 	Ui2	);
	TEST_ASSERT_EQUAL_INT( 	I1, 	I2	);
	TEST_ASSERT_EQUAL_INT( 	Di1, 	Di2	);
	TEST_ASSERT_EQUAL_INT(	Udi1, 	Udi2);

	TEST_DONE;
}

_TEST test_string(void)
{
	TEST_ASSERT_EQUAL_STRING(String1, String2 );

	TEST_DONE;
}

_TEST test_wstring(void)
{
	TEST_ASSERT_EQUAL_WSTRING(WString1,	WString2);

	TEST_DONE;
}

_TEST test_float(void)
{
	TEST_ASSERT_EQUAL_FLOAT(Real1, Real2);
	TEST_ASSERT_FLOAT_WITHIN(RealDeltaForComparison, Real1, Real2);

	TEST_ASSERT_EQUAL_REAL(Real1, Real2);
	TEST_ASSERT_REAL_WITHIN(RealDeltaForComparison, Real1, Real2);

	TEST_DONE;
}

_TEST test_double(void)
{
	TEST_ASSERT_EQUAL_DOUBLE(LReal1, LReal2);
	TEST_ASSERT_DOUBLE_WITHIN(LRealDeltaForComparison, LReal1, LReal2);

	TEST_ASSERT_EQUAL_LREAL(LReal1, LReal2);
	TEST_ASSERT_LREAL_WITHIN(LRealDeltaForComparison, LReal1, LReal2);

	TEST_DONE;
}

_TEST test_memory(void)
{
	TEST_ASSERT_EQUAL_MEM(Buffer1, Buffer2, sizeof(Buffer1)  );

	TEST_DONE;
}

_TEST test_null_true_and_false(void)
{
	TEST_ASSERT_NOT_NULL(Pointer);
	TEST_ASSERT_NOT_NULL(0); 	/* Not Ok */

	TEST_ASSERT_NULL(0); 		/* Ok */
	TEST_ASSERT_NULL(Pointer);

	Pointer = &Udi1;
	TEST_ASSERT_NULL(Pointer); /* Not Ok */

	TEST_DONE;
}

_TEST test_message(void)
{
	TEST_ASSERT_MESSAGE(ConditionFlag, "This text, if condition evaluates to false.");
	ConditionFlag = 0;
	TEST_ASSERT_MESSAGE(ConditionFlag, "This text, because condition evaluates to false.");
	ConditionFlag = 4;
	TEST_ASSERT_MESSAGE(ConditionFlag, "Nothing, as condition evaluates to true (!= 0).");

	TEST_DONE;
}

_TEST test_info(void)
{
	TEST_INFO("Info Text - for some comment");
	TEST_INFO_POS("Info Text - for some comment with position");

	TEST_DONE;
}

_TEST test_fail(void)
{
	TEST_FAIL("Always fails");

	TEST_DONE;
}

/*
B+R UnitTest: This is generated code.
Do not edit! Do not move!
Description: UnitTest Testprogramm infrastructure (TestSet).
LastUpdated: 2015-04-14 12:03:48Z
By B+R UnitTest Helper Version: 2.0.0.0
*/
UNITTEST_FIXTURES(fixtures)
{
	new_TestFixture("test_int", test_int),
	new_TestFixture("test_string", test_string),
	new_TestFixture("test_wstring", test_wstring),
	new_TestFixture("test_float", test_float),
	new_TestFixture("test_double", test_double),
	new_TestFixture("test_memory", test_memory),
	new_TestFixture("test_null_true_and_false", test_null_true_and_false),
	new_TestFixture("test_message", test_message),
	new_TestFixture("test_info", test_info),
	new_TestFixture("test_fail", test_fail),
};

UNITTEST_CALLER_COMPLETE_EXPLICIT(testSet_Asserts, "testSet_Asserts", setupTest, teardownTest, fixtures, 0, 0, 0);
```

#### testSuite.c
```c
/********************************************************************
 * COPYRIGHT -- Bernecker + Rainer
 ********************************************************************
 * Program: SPL_Asserts
 * Author: B+R
 ********************************************************************
 * Test registration and handshake
 ********************************************************************/

#include <bur/plctypes.h>

#ifdef _DEFAULT_INCLUDES
#include <AsDefault.h>
#endif

#include "UnitTest.h"

void _INIT initTestSuite(void)
{
	utInit(&Testsuite);
}

void _CYCLIC cyclicWithTest(void)
{
	/* Some code */
	utCyclic(&Testsuite);
}

void _EXIT exitTestSuite(void)
{
	utExit(&Testsuite);
}
```

### Program Logical/Infrastructure/TS_UnitTest/Samples/Framework_Features/SPL_Behavior (ANSIC) - This sample is about the control flow of test programs

#### TestBusy_AsyncronousVariables.var
```iecst
(********************************************************************
 * COPYRIGHT -- Bernecker + Rainer
 ********************************************************************
 * Program: SPL_Behavior
 * Author: B+R
 ********************************************************************
 * Local variables of program SPL_Behavior
 * For test sets in package TestBusy_Asyncronous
 ********************************************************************)
VAR
	GetMimeTypeResult : STRING[80] := '';
	webserverStatus : CfgGetWebServerStatus := (0);
	webserverGetMimeType : CfgGetWebMimeType := (0);
	webserverSetMimeType : CfgSetWebMimeType := (0);
END_VAR
```

#### iHelperFunction.h
```c
/********************************************************************
 * COPYRIGHT -- Bernecker + Rainer
 ********************************************************************
 * Program: SPL_Behavior
 * File: iHelperFunction.h
 * Author: B+R
 *******************************************************************/

#include <bur/plctypes.h>

#include "iPrototypes.h"

/* This Macro is for tracing the calls in the sample
(For exemplification)*/
#define LOG_FOR_EXEMPLIFICATION_CYCLIC_SET  \
	brsstrcat((UDINT)OutputString, (UDINT)"Cyclic set - "); \
	checkAndWriteCounterIfChanged(__LINE__, __FILE__); \
	CounterInSet++;

/* This Macro is for tracing the calls in the sample
(For exemplification)*/
#define LOG_FOR_EXEMPLIFICATION_TEST_CASE_1   \
	brsstrcat((UDINT)OutputString,(UDINT) "Call test 1 - "); \
	checkAndWriteCounterIfChanged(__LINE__, __FILE__);

/* This Macro is for tracing the calls in the sample
(For exemplification)*/
#define LOG_FOR_EXEMPLIFICATION_TEST_CASE_2 \
	brsstrcat((UDINT)OutputString,(UDINT) "Call test 2 - "); \
	checkAndWriteCounterIfChanged(__LINE__, __FILE__);

/* This Macro is for tracing the calls in the sample
(For exemplification)*/
#define LOG_FOR_EXEMPLIFICATION_TEST_CASE_3   \
	brsstrcat((UDINT)OutputString,(UDINT) "Call test 3 - "); \
	checkAndWriteCounterIfChanged(__LINE__, __FILE__);

/* This Macro is for tracing the calls in the sample
(For exemplification)*/
#define LOG_FOR_EXEMPLIFICATION_SETUP_SET  \
	brsstrcat((UDINT)OutputString, (UDINT)"Setup set - "); \
	checkAndWriteCounterIfChanged(__LINE__, __FILE__);

/* This Macro is for tracing the calls in the sample
(For exemplification)*/
#define LOG_FOR_EXEMPLIFICATION_TEARDOWN_SET  \
	brsstrcat((UDINT)OutputString, (UDINT)"Teardown set - "); \
	checkAndWriteCounterIfChanged(__LINE__, __FILE__);

 /* This Macro is for tracing the calls in the sample
(For exemplification)*/
#define LOG_FOR_EXEMPLIFICATION_SETUP_TEST \
	brsstrcat((UDINT)OutputString, (UDINT)"Setup test - "); \
	checkAndWriteCounterIfChanged(__LINE__, __FILE__);

/* This Macro is for tracing the calls in the sample
(For exemplification)*/
#define LOG_FOR_EXEMPLIFICATION_TEARDOWN_TEST  \
	brsstrcat((UDINT)OutputString, (UDINT)"Teardown test - "); \
	checkAndWriteCounterIfChanged(__LINE__, __FILE__);

/* ************************************************/

/* Add this line behind a LOG_FOR_EXEMPLIFICATION_TEST_CASE_x to simulate an asyncron test case
 This Macro is for tracing the calls in the sample
(For exemplification)*/
#define LOG_FOR_EXEMPLIFICATION_TEST_BUSY  if(CountTestCaseRuns < DEF_BUSY_STEPS)\
	{\
	countTestCaseRuns++; \
	brsstrcat((UDINT)OutputString,(UDINT) "TEST_BUSY (recall in next cycle) - "); \
	TEST_BUSY; } \
	else { CountTestCaseRuns = 0;}
```

#### iPrototypes.h
```c
/********************************************************************
 * COPYRIGHT -- Bernecker + Rainer
 ********************************************************************
 * Program: SPL_Behavior
 * File: iPrototypes.h
 * Author: B+R
 *******************************************************************/

#include <bur/plctypes.h>

/* Prototyping of functions  */
void 	resetDataForTestSet();
void 	checkAndWriteCounterIfChanged( unsigned long line, const char *file);

void	resetDataForTestSet_Complete();
void	resetDataForTestSet_TestCases();
void	resetDataForTestSet_SetSetupTeardown();
void	resetDataForTestSet_TestSetupTeardown();
```

#### iHelperFunction.c
```c
/********************************************************************
 * COPYRIGHT -- Bernecker + Rainer
 ********************************************************************
 * Program: SPL_Behavior
 * File: iHelperFunction.c
 * Author: B+R
 *******************************************************************/

#include <bur/plctypes.h>

#ifdef _DEFAULT_INCLUDES
#include <AsDefault.h>
#endif

#include "UnitTest.h"
#include "AsBrStr.h"
#include "iPrototypes.h"

void resetDataForTestSet()
{
	brsstrcpy((UDINT)OutputString, (UDINT)"");
	CounterInSet = 0;
	CounterInSet_LastChecked = -1;
	CounterToStringBuffer[0] = 0;
}

void checkAndWriteCounterIfChanged( unsigned long line, const char *file)
{
	if(CounterInSet_LastChecked != CounterInSet)
	{
		addFailure((char*)OutputString, line, file);

		CounterInSet_LastChecked = CounterInSet;
		brsitoa(CounterInSet + 1, (UDINT) CounterToStringBuffer);

		brsstrcpy((UDINT)OutputString, (UDINT)"( ");
		brsstrcat((UDINT)OutputString, (UDINT)CounterToStringBuffer);
		/*		brsstrcat((UDINT)OutputString, (UDINT)". task cylce in TestSet) "); */
		brsstrcat((UDINT)OutputString, (UDINT)". cylce) ");

		addFailure((char*)OutputString, line, file);

	}
	else if(OutputString[0])
	{
		/*		TEST_FAIL(OutputString);*/
		addFailure((char*)OutputString, line, file);
	}

}
```

#### README.txt
```
Please note

The samples in this program provides no good programming style!
They are solely for demonstrating the behavior of the framework.
Bad style:
	o	Asserts should only be used to verify the test case as the report should be short ans meaningful (No explainings, just the relevant facts).
	o	Asserts should only be used in test cases.
	o	Test cases should be named meaningful.
	o	Macros are used instead of helper functions.
```

#### testSuite.c
```c
/********************************************************************
 * COPYRIGHT -- Bernecker + Rainer
 ********************************************************************
 * Program: SPL_Behavior
 * Author: B+R
 ********************************************************************
 * Test registration and handshake
 ********************************************************************/

#include <bur/plctypes.h>

#ifdef _DEFAULT_INCLUDES
#include <AsDefault.h>
#endif

#include "UnitTest.h"

#include "iPrototypes.h"

void _INIT initTestSuite(void)
{
	utInit(&Testsuite);
}

void _CYCLIC cyclicWithTest(void)
{
	/* Some code */
	utCyclic(&Testsuite);

	if(Testsuite.TestFinishedDone)
	{
		resetDataForTestSet_Complete();
		resetDataForTestSet_TestCases();
		resetDataForTestSet_SetSetupTeardown();
		resetDataForTestSet_TestSetupTeardown();
	}
}

void _EXIT exitTestSuite(void)
{
	utExit(&Testsuite);
}
```

#### test_SetTestCases_TestSetup_TestTeardown.c
```c
/********************************************************************
* COPYRIGHT -- Bernecker + Rainer
********************************************************************
* Program: SPL_Behavior
* Author: B+R
********************************************************************
* This test set shows the sequence of calls within a test set
* Add some busy conditions or test cases to see the changes.
********************************************************************/

#include <bur/plctypes.h>

#ifdef _DEFAULT_INCLUDES
#include <AsDefault.h>
#endif

#include "UnitTest.h"

#include "iHelperFunction.h"

void resetDataForTestSet_TestSetupTeardown()
{
	resetDataForTestSet();
}

_CYCLIC_SET(void)
{
	LOG_FOR_EXEMPLIFICATION_CYCLIC_SET;
	return;
}

_SETUP_TEST(void)
{
	LOG_FOR_EXEMPLIFICATION_SETUP_TEST;
	TEST_DONE;
}

_TEARDOWN_TEST(void)
{
	LOG_FOR_EXEMPLIFICATION_TEARDOWN_TEST;
	TEST_DONE;
}

_TEST test_1(void)
{
	LOG_FOR_EXEMPLIFICATION_TEST_CASE_1;
	TEST_DONE;
}

_TEST test_2(void)
{
	LOG_FOR_EXEMPLIFICATION_TEST_CASE_2;
	TEST_DONE;
}

_TEST test_3(void)
{
	LOG_FOR_EXEMPLIFICATION_TEST_CASE_3;
	TEST_DONE;
}

/*
B+R UnitTest: This is generated code.
Do not edit! Do not move!
Description: UnitTest Testprogramm infrastructure (TestSet).
LastUpdated: 2015-04-14 12:03:48Z
By B+R UnitTest Helper Version: 2.0.0.0
*/
UNITTEST_FIXTURES(fixtures)
{
	new_TestFixture("test_1", test_1),
	new_TestFixture("test_2", test_2),
	new_TestFixture("test_3", test_3),
};

UNITTEST_CALLER_COMPLETE_EXPLICIT(test_SetTestCases_TestSetup_TestTeardown, "test_SetTestCases_TestSetup_TestTeardown", setupTest, teardownTest, fixtures, 0, 0, cyclicSetCaller);
```

#### TestBusy_Asyncronous.c
```c
/********************************************************************
* COPYRIGHT -- Bernecker + Rainer
********************************************************************
* Program: SPL_Behavior
* Author: B+R
********************************************************************
* This test set shows the option to call a function
*       (test case, setup or teardown) until "done".
* This is usable for example for testing asynchronous FUBs.
********************************************************************/

#include <bur/plctypes.h>

#ifdef _DEFAULT_INCLUDES
#include <AsDefault.h>
#endif

#include "AsArCfg.h"

#include "UnitTest.h"

/* _SETUP_TEST() is called before each test case of this test set */
_SETUP_TEST(void)
{
	/* Call */
	webserverStatus.enable = 0;
	CfgGetWebServerStatus(&webserverStatus);

	webserverSetMimeType.enable = 0;
	CfgSetWebMimeType(&webserverSetMimeType);

	webserverGetMimeType.enable = 0;
	CfgGetWebMimeType(&webserverGetMimeType);

	/* Done */
	TEST_DONE;
}

/* _TEARDOWN_SET() is called at end of this test set */
_TEARDOWN_SET(void)
{
	/* Call */
	webserverStatus.enable = 0;
	CfgGetWebServerStatus(&webserverStatus);

	webserverSetMimeType.enable = 0;
	CfgSetWebMimeType(&webserverSetMimeType);

	webserverGetMimeType.enable = 0;
	CfgGetWebMimeType(&webserverGetMimeType);

	/* Done */
	TEST_DONE;
}

/* Sample test case tests async. FB CfgGetWebServerStatus() */
_TEST test_AsyncFub(void)
{
	/* Call */
	webserverStatus.enable = 1;
	CfgGetWebServerStatus(&webserverStatus);

	/* Wait  */
	TEST_BUSY_CONDITION(ERR_FUB_BUSY == webserverStatus.status );

	/* Test */
	TEST_ASSERT_EQUAL_INT( ERR_OK, webserverStatus.status  );
	TEST_ASSERT_EQUAL_INT(cfgWEB_MODE_ENABLED,  webserverStatus.mode);

	/* Done */
	TEST_DONE;
}

/* Sample test case tests async. FB CfgGetWebMimeType() */
_TEST test_getMimeType(void)
{
	/* Call */
	webserverGetMimeType.enable = 1;
	webserverGetMimeType.pFileExtension =  (UDINT) "*.txt";
	webserverGetMimeType.pMimeType = (UDINT)GetMimeTypeResult;
	webserverGetMimeType.len = sizeof(GetMimeTypeResult) - 1;
	CfgGetWebMimeType(&webserverGetMimeType);

	/* Wait  */
	TEST_BUSY_CONDITION_MSG(ERR_FUB_BUSY == webserverGetMimeType.status,  "Fub is busy");

	/* Test */
	TEST_ASSERT_EQUAL_INT( ERR_OK, webserverGetMimeType.status  );
	TEST_ASSERT_EQUAL_STRING("text/plain", GetMimeTypeResult   );

	/* Done */
	TEST_DONE;
}

/*
B+R UnitTest: This is generated code.
Do not edit! Do not move!
Description: UnitTest Testprogramm infrastructure (TestSet).
LastUpdated: 2015-04-14 12:03:48Z
By B+R UnitTest Helper Version: 2.0.0.0
*/
UNITTEST_FIXTURES(fixtures)
{
	new_TestFixture("test_AsyncFub", test_AsyncFub),
	new_TestFixture("test_getMimeType", test_getMimeType),
};

UNITTEST_CALLER_COMPLETE_EXPLICIT(TestBusy_Asyncronous, "TestBusy_Asyncronous", setupTest, 0, fixtures, 0, teardownSet, 0);
```

#### TestBusy_Asyncronous_with_CyclicSet.c - This test set adds additional information to the test report (for illustration only)
```c
/********************************************************************
* COPYRIGHT -- Bernecker + Rainer
********************************************************************
* Program: SPL_Behavior
* Author: B+R
********************************************************************
* This test set shows the option to call a function
*       (test case, setup or teardown) until "done".
* This is usable for example for testing asynchronous FUBs.
********************************************************************/

#include <bur/plctypes.h>

#ifdef _DEFAULT_INCLUDES
#include <AsDefault.h>
#endif

#include "UnitTest.h"

#include "iHelperFunction.h"

/*_CYCLIC_SET() is called in each cycle as long this Test Set is the active test set*/
_CYCLIC_SET(void)
{
	LOG_FOR_EXEMPLIFICATION_CYCLIC_SET;
	CfgGetWebServerStatus(&webserverStatus);
	CfgSetWebMimeType(&webserverSetMimeType);
	CfgGetWebMimeType(&webserverGetMimeType);

}

/* _SETUP_SET() is called at the beginning of this test set */
_SETUP_SET(void)
{
	resetDataForTestSet();

	LOG_FOR_EXEMPLIFICATION_SETUP_SET;

	/*Disable FB at beginning of this test set*/
	webserverStatus.enable = 0;
	webserverSetMimeType.enable = 0;
	webserverGetMimeType.enable = 0;

	TEST_DONE;
}

/* _SETUP_TEST() is called before each test case of this test set */
_SETUP_TEST(void)
{
	LOG_FOR_EXEMPLIFICATION_SETUP_TEST;

	/*Disable FB at beginning of this test set*/
	webserverStatus.enable = 0;
	webserverSetMimeType.enable = 0;
	webserverGetMimeType.enable = 0;

	TEST_DONE;
}

/* _TEARDOWN_SET() is called at end of this test set */
_TEARDOWN_SET(void)
{
	LOG_FOR_EXEMPLIFICATION_TEARDOWN_SET;
	/*Disable FB after each test case*/
	webserverStatus.enable = 0;
	webserverSetMimeType.enable = 0;
	webserverGetMimeType.enable = 0;

	/* Done */
	TEST_DONE;
}

/* Sample test case tests async. FB CfgGetWebServerStatus() */
_TEST test_AsyncFub(void)
{
	LOG_FOR_EXEMPLIFICATION_TEST_CASE_1;

	/*Silent  wait  as FB is still busy*/
	TEST_BUSY_CONDITION(ERR_FUB_BUSY == webserverStatus.status  );

	webserverStatus.enable = 1;

	/*Silent  wait  as FB is not yet enabled*/
	TEST_BUSY_CONDITION( ERR_FUB_ENABLE_FALSE == webserverStatus.status );

	/* Test */
	TEST_ASSERT_EQUAL_INT( ERR_OK, webserverStatus.status  );
	TEST_ASSERT_EQUAL_INT(cfgWEB_MODE_ENABLED,  webserverStatus.mode);

	/* Done */
	TEST_DONE;
}

/* Sample test case tests async. FB CfgGetWebMimeType() */
_TEST test_getMimeType(void)
{
	LOG_FOR_EXEMPLIFICATION_TEST_CASE_3;

	TEST_BUSY_CONDITION_MSG(ERR_FUB_BUSY == webserverGetMimeType.status,  "Fub is busy");

	webserverGetMimeType.enable = 1;
	webserverGetMimeType.pFileExtension =  (UDINT) "*.txt";
	webserverGetMimeType.pMimeType = (UDINT)GetMimeTypeResult;
	webserverGetMimeType.len = sizeof(GetMimeTypeResult) - 1;

	/* Wait  */
	TEST_BUSY_CONDITION_MSG(ERR_FUB_ENABLE_FALSE == webserverGetMimeType.status,  "Fub is not enabled");

	/* Test */
	TEST_ASSERT_EQUAL_INT( ERR_OK, webserverGetMimeType.status  );
	TEST_ASSERT_EQUAL_STRING("text/plain", GetMimeTypeResult   );

	/* Done */
	TEST_DONE;
}

/*
B+R UnitTest: This is generated code.
Do not edit! Do not move!
Description: UnitTest Testprogramm infrastructure (TestSet).
LastUpdated: 2015-04-14 12:03:48Z
By B+R UnitTest Helper Version: 2.0.0.0
*/
UNITTEST_FIXTURES(fixtures)
{
	new_TestFixture("test_AsyncFub", test_AsyncFub),
	new_TestFixture("test_getMimeType", test_getMimeType),
};

UNITTEST_CALLER_COMPLETE_EXPLICIT(TestBusy_Asyncronous_with_CyclicSet, "TestBusy_Asyncronous_with_CyclicSet", setupTest, 0, fixtures, setupSet, teardownSet, cyclicSetCaller);
```

### Package Logical/Infrastructure/TS_UnitTest/Templates/HelperTool_Supported - Easy mode: focus on writing tests

### Package Logical/Infrastructure/TS_UnitTest/Templates/HelperTool_Supported/TestSet_Templates - Multiple variants of valid test sets

### Set_Complete.c
```c
/********************************************************************
 * COPYRIGHT --
 ********************************************************************
 * Program: -
 * Author:
 * Created:
 ********************************************************************
 * Tests for ...
 ********************************************************************/

#include <bur/plctypes.h>

#ifdef _DEFAULT_INCLUDES
#include <AsDefault.h>
#endif

#include "UnitTest.h"

_CYCLIC_SET()
{

	/* TODO:  add code running cyclically while test set is active here */
	return;
}

_SETUP_SET(void)
{
	/* TODO:  add code running before test set here */
	TEST_DONE;
}

_TEARDOWN_SET(void)
{
	/* TODO:  add code running after test set here */
	TEST_DONE;
}

_SETUP_TEST(void)
{
	/* TODO:  add code running before test case here */
	TEST_DONE;
}

_TEARDOWN_TEST(void)
{
	/* TODO:  add code running after test case here */
	TEST_DONE;
}

_TEST testcase1(void)
{

	/* TODO:  add assertions here */

	/* test is done */
	TEST_DONE;
}
```

### Package Logical/Infrastructure/TS_UnitTest/Templates/NoToolSupport - Advanced mode: more control over fixtures

### Program Logical/Infrastructure/TS_UnitTest/Templates/NoToolSupport/utTemplate_manual (ANSIC) - Empty Template without support of helper tool

#### FixtureOfTestSets.c
```c
/********************************************************************
 * COPYRIGHT --
 ********************************************************************
 * Program: -
 * Author:
 * Created:
 ********************************************************************
 * Test Set Fixture
 ********************************************************************/

#include "UnitTest.h"

/* TODO: Add your sets here

UNITTEST_TESTSET_DECLARATION testSet1;
UNITTEST_TESTSET_DECLARATION testSet2;
*/

/* List of all test sets of the test programm
they will be executed in the given order*/
UNITTEST_TESTSET_FIXTURES (utTestSets)
{
#warning TODO: Add your sets here
	/* TODO: Add your sets here
	new_TestSet(testSet1),
	new_TestSet(testSet2)*/
	{
		0
	} /* Place holder for test sets, can be removed */
};

/*Handler of test set list */
UNTITTEST_TESTSET_HANDLER();
```

#### testSuite.c
```c
/********************************************************************
 * COPYRIGHT --
 ********************************************************************
 * Program: -
 * Author:
 * Created:
 ********************************************************************
 * Test registration and handshake
 ********************************************************************/

#include <bur/plctypes.h>

#ifdef _DEFAULT_INCLUDES
#include <AsDefault.h>
#endif

#include "UnitTest.h"

void _INIT initTestSuite(void)
{
	utInit(&Testsuite);
}

void _CYCLIC cyclicWithTest(void)
{
	utCyclic(&Testsuite);
}

void _EXIT exitTestSuite(void)
{
	utExit(&Testsuite);
}
```

### Package Logical/Infrastructure/TS_UnitTest/Templates/NoToolSupport/TestSet_Templates - Multiple variants of valid test sets

### Set_Complete.c
```c
/********************************************************************
 * COPYRIGHT --
 ********************************************************************
 * Program: -
 * Author:
 * Created:
 ********************************************************************
 * Tests for ...
 ********************************************************************/

#include <bur/plctypes.h>

#ifdef _DEFAULT_INCLUDES
#include <AsDefault.h>
#endif

#include "UnitTest.h"

/* called when test set is active. */
_CYCLIC_SET()
{

	/* TODO:  add code running cyclically while test set is active here */
	return;
}

/* called before first test case of test set*/
_SETUP_SET(void)
{
	/* TODO:  add code running before test set here */
	TEST_DONE;
}

/* called after last test case of test set */
_TEARDOWN_SET(void)
{
	/* TODO:  add code running after test set here */
	TEST_DONE;
}

/* called before a test case first called */
_SETUP_TEST(void)
{
	/* TODO:  add code running before test case here */
	TEST_DONE;
}

/* called after a test case is done*/
_TEARDOWN_TEST(void)
{
	/* TODO:  add code running after test case here */
	TEST_DONE;
}
/* ---------------------------*/

/* a test case*/
_TEST testcase1(void)
{

	/* TODO:  add assertions here */

	/* test is done */
	TEST_DONE;
}

/* a test case*/
_TEST testcase2(void)
{
	/* TODO:  add assertions here */

	/* test is done */
	TEST_DONE;
}

#warning TODO: Add your test cases here
/*TODO: Add your test cases here */
UNITTEST_FIXTURES(fixtures)
{
	new_TestFixture("testcase1",testcase1),
	                new_TestFixture("testcase2",testcase2),
};

#warning TODO: rename testset (Param 1 and 2)
UNITTEST_CALLER_COMPLETE(testSetComplete, "testSetComplete",fixtures);
```

### Set_Testcases.c
```c
/********************************************************************
 * COPYRIGHT --
 ********************************************************************
 * Program: -
 * Author:
 * Created:
 ********************************************************************
 * Tests for ...
 ********************************************************************/

#include <bur/plctypes.h>

#ifdef _DEFAULT_INCLUDES
#include <AsDefault.h>
#endif

#include "UnitTest.h"

/* a test case*/
_TEST testcase1(void)
{

	/* TODO: add assertions here */

	/* test is done */
	TEST_DONE;
}

/* a test case*/
_TEST testcase2(void)
{
	/* TODO: add assertions here */

	/* test is done */
	TEST_DONE;
}

#warning TODO: Add your test cases here
/*TODO: Add your test cases here */
UNITTEST_FIXTURES(fixtures)
{
	new_TestFixture("testcase1",testcase1),
	                new_TestFixture("testcase2",testcase2),
};

#warning TODO: rename testset (Param 1 and 2)
UNITTEST_CALLER_TEST(testSet_testcases, "testSet_testcases",fixtures);
```

### UsbMgr.typ
```iecst
(*Structure types*)

TYPE
	DevLink_FUBType : 	STRUCT  (*Contains all FileIO function blocks*)
		UsbNodeListGet_0 : UsbNodeListGet; (*UsbNoteListGet instance*)
		UsbNodeGet_0 : UsbNodeGet; (*UsbNodeGet instance*)
		UsbMsDeviceReady_0 : UsbMsDeviceReady; (*UsbMsDeviceReady instance*)
		DevLink_0 : DevLink; (*DevLink instance*)
		DevUnlink_0 : DevUnlink; (*DevUnlink instance*)
	END_STRUCT;
	DevLinkControlType : 	STRUCT  (*Control structure which contains everything necessary for the file handling machine*)
		Step : StepType; (*Current step*)
		Commands : UsbCommandsType; (*Commands*)
		Parameters : UsbParametersType; (*Parameters*)
		FUB : DevLink_FUBType; (*All FileIO FUBs*)
	END_STRUCT;
	UsbCommandsType : 	STRUCT  (*USB commands structure*)
		GetUSBList : BOOL; (*Get usb list *)
		GetUSBInfo : BOOL; (*Get usb info*)
		DevLink : BOOL; (*Devlink*)
		DevUnlink : BOOL; (*Devunlink*)
		ErrAck : BOOL; (*Acknowledge error*)
	END_STRUCT;
	UsbParametersType : 	STRUCT  (*USB parameters structure*)
		ErrorID : UINT; (*FUB error ID*)
		NodeList : ARRAY[0..MAX_IDX_USB_DEV_LIST]OF UDINT; (*List of connected usb devices*)
		NodeInfoList : ARRAY[0..MAX_IDX_USB_DEV_LIST]OF usbNode_typ; (*Buffer for usb info*)
		FileDevName : ARRAY[0..MAX_IDX_USB_DEV_LIST]OF STRING[30]; (*File device names*)
		FileDevHandle : ARRAY[0..MAX_IDX_USB_DEV_LIST]OF UDINT; (*File device handle (needed for unlinking the device)*)
		LinkParam : STRING[30]; (*Parameter string to link a device*)
		Index : USINT; (*List index*)
	END_STRUCT;
END_TYPE

(*Enumerations*)

TYPE
	StepType :
		( (*Enumeration of the possible machine states*)
		STATE_WAIT := 0, (*Wait state*)
		STATE_GET_USB_LIST, (*Getting list of usb devices*)
		STATE_GET_USB_INFO, (*Getting info from a usb device*)
		STATE_DEV_LINK, (*Linking device*)
		STATE_DEV_UNLINK, (*Unlinking device*)
		STATE_ERROR_USB (*Some FUB returned an error*)
		);
END_TYPE
```

### Program Logical/Infrastructure/UserX/UserXMgr

#### UserXMgr.st
```iecst
//***********************************************************************
// Copyright: B&R Industrial Automation GmbH
// Author: B&R Industrial Automation GmbH
// Created: April 12, 2022
// Description: Tasks for user management.
//***********************************************************************

PROGRAM _INIT

	// Create folder for this component on the user file device
	DirCreate_0(enable := TRUE, pDevice := ADR('UserPartition'), pName := ADR(LOCAL_FOLDER));

	// Check if folder already exist and if so disabled the function block call
	IF DirCreate_0.status = fiERR_DIR_ALREADY_EXIST THEN
		DirCreate_0(enable := FALSE);
	END_IF

	// Initialize mapp function blocks
	UserXMgrUIConnect.User.Create.Lock := FALSE;
	UserXMgrUIConnect.User.Lock := FALSE;
	UserXMgrUIConnect.User.Edit.Lock := FALSE;
    UserXMgrUIConnect.User.Create.Dialog.UserName := "";
    UserXMgrUIConnect.User.Create.Dialog.NewPassword := "";
	UserXMgrUIConnect.User.Create.Dialog.ConfirmPassword := "";
	UserXMgrUIConnect.User.List.MaxSelection := USER_LIST_MAX_SELECTION;
	UserXMgrUIConnect.User.List.RangeStart := USER_LIST_RANGE_START;
	UserXMgrUIConnect.User.List.RangeEnd := USER_LIST_RANGE_END;
    MpUserXManagerUI_0.MpLink := ADR(gMpLinkUserXLogin);
    MpUserXManagerUI_0.Enable := TRUE;
    MpUserXManagerUI_0.UIConnect := ADR(UserXMgrUIConnect);
	MpUserXManagerUI_0();

	MpUserXLoginUI_0.MpLink := ADR(gMpLinkUserXLogin);
    MpUserXLoginUI_0.Enable := TRUE;
	MpUserXLoginUI_0.UIConnect := ADR(UserXLoginUIConnect);
	MpUserXLoginUI_0();

	MpUserXLogin_0.MpLink := ADR(gMpLinkUserXLogin);
	MpUserXLogin_0.Enable := TRUE;
	MpUserXLogin_0();

END_PROGRAM

PROGRAM _CYCLIC

	// Error reset
	IF NOT MpUserXManagerUI_0.Error THEN
		MpUserXManagerUI_0.ErrorReset := FALSE;
    END_IF

	IF NOT MpUserXLoginUI_0.Error THEN
		MpUserXLoginUI_0.ErrorReset := FALSE;
    END_IF

	IF NOT MpUserXLogin_0.Error THEN
		MpUserXLogin_0.ErrorReset := FALSE;
    END_IF

	// Assign MpLinks
	MpUserXManagerUI_0.MpLink := ADR(gMpLinkUserXLogin);
	MpUserXLoginUI_0.MpLink := ADR(gMpLinkUserXLogin);
	MpUserXLogin_0.MpLink := ADR(gMpLinkUserXLogin);

	// Call function blocks
	MpUserXManagerUI_0();
	MpUserXLoginUI_0();
	MpUserXLogin_0();

END_PROGRAM

PROGRAM _EXIT

	// Disable the function blocls to unlink the MpLinks
    MpUserXManagerUI_0.Enable := FALSE;
	MpUserXLoginUI_0.Enable := FALSE;
	MpUserXLogin_0.Enable := FALSE;

	// Call function blocks
	MpUserXManagerUI_0();
	MpUserXLoginUI_0();
	MpUserXLogin_0();

END_PROGRAM
```

### AsMem.var
```iecst
VAR CONSTANT
	asmemERR_DESTROY	: UINT	:= 30501;		(*cannot free up memory partition*)
	asmemERR_CREATE	: UINT	:= 30500;			(*cannot create memory partition*)
	asmemERR_NOMEM	: UINT	:= 30502;			(*cannot allocate memory block with requested size*)
	asmemERR_INFO	: UINT	:= 30504;			(*information about free memory can not be detected*)
	asmemERR_FREE	: UINT	:= 30503;			(*cannot free up memory block*)
END_VAR
```

### Library Logical/Libraries/Gat (IEC)
Depends on: ArCfgMan, IoMapMan

#### Types.typ - Exported data types
```iecst
TYPE
	GatIoForcHandInternalType : 	STRUCT
		AsIOSetForceValue_Int : AsIOSetForceValue;
		AsIODisableForcing_Int : AsIODisableForcing;
		AsIOEnableForcing_Int : AsIOEnableForcing;
		AsIODPStatus_Int : AsIODPStatus;
		IO_OpenIoMap_Int : IO_OpenIoMap;
		IO_CloseIoMap_Int : IO_CloseIoMap;
		AR_OpenArCfg_Int : AR_OpenArCfg;
		AR_CloseArCfg_Int : AR_CloseArCfg;
		ForceValue : ARRAY[0..gatMAX_IDX_IO_MODULES,0..gatMAX_IDX_IO_CHANNELS]OF UDINT;
		ForceEnabled : ARRAY[0..gatMAX_IDX_IO_MODULES,0..gatMAX_IDX_IO_CHANNELS]OF BOOL;
		IoMapIdent : UDINT;
		ArCfgIdent : UDINT;
		IdxModuleNames : UDINT;
		IdxModule : UDINT;
		IdxIoChannel : UDINT;
		IdxModuleCmd : UDINT;
		IdxIoChannelCmd : UDINT;
		NrOfModules : UDINT;
		NrOfIoChannels : UDINT;
		TempChannel : GatIoChannelType;
		CommandState : USINT;
		InitState : USINT;
	END_STRUCT;
	GatIoForceType : 	STRUCT  (*Structure for forcing an IO value*)
		ActualValue : UDINT; (*Actual value on the physical channel*)
		ForceValue : UDINT; (*Force value*)
		SetForceActive : BOOL; (*TRUE: force value is used; FALSE: actual value is used*)
		DpName : STRING[100]; (*IO data point name*)
		RefreshActualValue : BOOL;
	END_STRUCT;
	GatIoMapType : 	STRUCT  (*Structure to read the io map channels*)
		NumberOfChannels : UDINT; (*Number of available IO channels*)
		Ident : UDINT; (*IO map ident*)
	END_STRUCT;
	GatIoChannelType : 	STRUCT  (*Io channel information*)
		Type : IO_Type_enum;
		Inverted : BOOL;
		ChannelName : STRING[80];
		PvName : STRING[80];
		ModulePath : STRING[80];
		TaskClass : USINT;
		IoForcing : GatIoForceType;
	END_STRUCT;
	GatIoModulesType : 	STRUCT
		ModuleName : STRING[80];
		ModulePath : STRING[80];
		IoChannels : ARRAY[0..gatMAX_IDX_IO_CHANNELS]OF GatIoChannelType;
		NrOfIoChannels : USINT;
	END_STRUCT;
END_TYPE
```

#### Constants.var - Exported constants
```iecst
VAR CONSTANT
	gatMAX_IDX_IO_CHANNELS : USINT := 31;
	gatMAX_IDX_IO_MODULES : USINT := 19;
	CONST_PI : REAL := 3.14159265359;
END_VAR
```

#### Gat.fun - Exported functions and function blocks
```iecst
{REDUND_ERROR} FUNCTION GatDegreeToDistance : REAL (*This function translates a given degree and radius to the corresponding length on a linear axis*) (*$GROUP=User,$CAT=User,$GROUPICON=User.png,$CATICON=User.png*)
	VAR_INPUT
		Degree : REAL;
		Radius : REAL;
	END_VAR
END_FUNCTION

FUNCTION_BLOCK GatIoForcingHandler
	VAR_INPUT
		Enable : BOOL; (*Enable of function block*)
		IoModules : REFERENCE TO ARRAY[0..gatMAX_IDX_IO_MODULES] OF GatIoModulesType; (*Reference to Module array*)
		SelectedRefreshMode : BOOL; (*Optional: Only selecteded channels will be refreshed: Depending on the number of IO channels in the project, this may greatly improve the performance*)
		ResetAllForcing : BOOL; (*Reset forcing on all io channels*)
	END_VAR
	VAR_OUTPUT
		Initializing : BOOL; (*Function block is initializing the module and Io structure*)
		Ready : BOOL; (*Initialization is complete, Io channels can be forced now*)
		CommandBusy : BOOL; (*Command is busy*)
		CommandDone : BOOL; (*Command is done*)
	END_VAR
	VAR
		Internal : GatIoForcHandInternalType;
	END_VAR
END_FUNCTION_BLOCK

FUNCTION GatIoIsVisible : BOOL
	VAR_INPUT
		ChannelName : REFERENCE TO STRING[80];
	END_VAR
END_FUNCTION

{REDUND_ERROR} FUNCTION GatMakeIoDpName : BOOL (*Creates the IO data point name from the given information*) (*$GROUP=User,$CAT=User,$GROUPICON=User.png,$CATICON=User.png*)
	VAR_INPUT
		IoChannel : GatIoChannelType;
		DpName : REFERENCE TO STRING[100];
	END_VAR
END_FUNCTION
```

#### GatDegreeToDistance.st
```iecst
// This function translates a given degree and radius to the corresponding length on a linear axis
FUNCTION GatDegreeToDistance
	GatDegreeToDistance := (Degree / 360.0) * 2.0 * CONST_PI * Radius;
END_FUNCTION
```

#### GatIoForcingHandler.st
```iecst
//*********************************************************************************
//* Copyright: B&R Industrial Automation GmbH
//* Created:   27 July, 2021/16:41
//* Handles Io forcing
//********************************************************************************

// Handles IO forcing for all modules
FUNCTION_BLOCK GatIoForcingHandler
	// Function block not enabled
	IF NOT Enable THEN
		// Close arcfg
		IF Internal.ArCfgIdent <> 0 THEN
			Internal.AR_CloseArCfg_Int.Ident := Internal.ArCfgIdent;
			Internal.AR_CloseArCfg_Int.Enable := TRUE;
			Internal.AR_CloseArCfg_Int.Store := FALSE;
			Internal.AR_CloseArCfg_Int();
			IF Internal.AR_CloseArCfg_Int.Status = ERR_OK THEN
				Internal.AR_CloseArCfg_Int.Enable := FALSE;
				Internal.AR_CloseArCfg_Int.Store := FALSE;
				Internal.AR_CloseArCfg_Int();
				Internal.ArCfgIdent := 0;
			END_IF
		END_IF
		// Close iomap
		IF Internal.IoMapIdent <> 0 THEN
			Internal.IO_CloseIoMap_Int.Ident := Internal.IoMapIdent;
			Internal.IO_CloseIoMap_Int.Enable := TRUE;
			Internal.IO_CloseIoMap_Int.Store := FALSE;
			Internal.IO_CloseIoMap_Int();
			IF Internal.IO_CloseIoMap_Int.Status = ERR_OK THEN
				Internal.IO_CloseIoMap_Int.Enable := FALSE;
				Internal.IO_CloseIoMap_Int.Store := FALSE;
				Internal.IO_CloseIoMap_Int();
				Internal.IoMapIdent := 0;
			END_IF
		END_IF
		// Function block disabled, return here
		Internal.InitState := 0;
		Internal.CommandState := 0;
		Internal.NrOfIoChannels := 0;
		Internal.NrOfModules := 0;
		Initializing := FALSE;
		Ready := FALSE;
		RETURN;
	END_IF

	// Initialize Io module and channel structure
	IF NOT Ready THEN
		Initializing := TRUE;
		// Open arcfg
		IF Internal.ArCfgIdent = 0 THEN
			Internal.InitState := 0;
			Internal.AR_OpenArCfg_Int.Enable := TRUE;
			Internal.AR_OpenArCfg_Int();
			IF Internal.AR_OpenArCfg_Int.Status = ERR_OK THEN
				Internal.ArCfgIdent := Internal.AR_OpenArCfg_Int.Ident;
				Internal.NrOfModules := AR_NumberOfModules(Internal.ArCfgIdent);
				Internal.AR_OpenArCfg_Int.Enable := FALSE;
				Internal.AR_OpenArCfg_Int();
			ELSE
				RETURN;
			END_IF
		END_IF
		// Open iomap
		IF Internal.IoMapIdent = 0 THEN
			Internal.InitState := 0;
			Internal.IO_OpenIoMap_Int.Enable := TRUE;
			Internal.IO_OpenIoMap_Int();
			IF Internal.IO_OpenIoMap_Int.Status = ERR_OK THEN
				Internal.IdxIoChannel := 1;
				Internal.IoMapIdent := Internal.IO_OpenIoMap_Int.Ident;
				Internal.NrOfIoChannels := Internal.IO_OpenIoMap_Int.NumberOfChannels;
				Internal.IO_OpenIoMap_Int.Enable := FALSE;
				Internal.IO_OpenIoMap_Int();
				brsmemset(ADR(IoModules), 0, SIZEOF(IoModules));
			ELSE
				RETURN;
			END_IF
		END_IF

		// iomap and arcfg are open, start initialization
		CASE Internal.InitState OF
			0: // Find all visible IoChannels and sort them by module path
				// Loop through IoChannels
				IF IO_ReadChannel(Internal.IoMapIdent, Internal.IdxIoChannel, ADR(Internal.TempChannel.Type), ADR(Internal.TempChannel.Inverted),
					ADR(Internal.TempChannel.ChannelName), ADR(Internal.TempChannel.PvName), ADR(Internal.TempChannel.ModulePath), ADR(Internal.TempChannel.TaskClass)) THEN
					// Check visibility
					IF (NOT GatIoIsVisible(ADR(Internal.TempChannel.ChannelName))) OR (brsstrlen(ADR(Internal.TempChannel.ModulePath)) = 0) THEN
						Internal.IdxIoChannel := Internal.IdxIoChannel + 1;
						IF Internal.IdxIoChannel > Internal.NrOfIoChannels THEN
							Internal.InitState := Internal.InitState + 1;
							Internal.IdxModule := 0;
						END_IF
						RETURN;
					END_IF
					// Search related module
					FOR Internal.IdxModule := 0 TO gatMAX_IDX_IO_MODULES DO
						IF brsstrcmp(ADR(IoModules[Internal.IdxModule].ModulePath), ADR('')) = 0 THEN
							// Related module not in list yet, add module
							brsstrcpy(ADR(IoModules[Internal.IdxModule].ModulePath), ADR(Internal.TempChannel.ModulePath));
						END_IF
						IF brsstrcmp(ADR(IoModules[Internal.IdxModule].ModulePath), ADR(Internal.TempChannel.ModulePath)) = 0 THEN
							// Module found
							GatMakeIoDpName(Internal.TempChannel, ADR(Internal.TempChannel.IoForcing.DpName));
							IoModules[Internal.IdxModule].IoChannels[IoModules[Internal.IdxModule].NrOfIoChannels] := Internal.TempChannel;
							IoModules[Internal.IdxModule].NrOfIoChannels := IoModules[Internal.IdxModule].NrOfIoChannels + 1;
							Internal.IdxIoChannel := Internal.IdxIoChannel + 1;
							IF Internal.IdxIoChannel > Internal.NrOfIoChannels THEN
								Internal.InitState := Internal.InitState + 1;
								Internal.IdxModule := 0;
							END_IF
							RETURN;
						END_IF
					END_FOR
				END_IF

			1: // Add Module names to each io module
				// Check if module index is populated
				IF brsstrlen(ADR(IoModules[Internal.IdxModule].ModulePath)) = 0 THEN
					Internal.IdxModule := Internal.IdxModule + 1;
					IF Internal.IdxModule > gatMAX_IDX_IO_MODULES THEN
						Internal.IdxModule := 0;
						Internal.IdxIoChannel := 0;
						Internal.InitState := Internal.InitState + 1;
					END_IF
					RETURN;
				END_IF
				// Loop through modules in arcfg to find the correct name
				FOR Internal.IdxModuleNames := 1 TO Internal.NrOfModules DO
					AR_GetModuleInfo(Internal.ArCfgIdent, Internal.IdxModuleNames, ADR(IoModules[Internal.IdxModule].ModuleName), ADR(IoModules[Internal.IdxModule].ModulePath));
					IF brsstrcmp(ADR(IoModules[Internal.IdxModule].ModulePath), ADR(IoModules[Internal.IdxModule].IoChannels[0].ModulePath)) = 0 THEN
						// Correct name was found
						Internal.IdxModule := Internal.IdxModule + 1;
						IF Internal.IdxModule > gatMAX_IDX_IO_MODULES THEN
							Internal.IdxModule := 0;
							Internal.IdxIoChannel := 0;
							Internal.InitState := Internal.InitState + 1;
						END_IF
						RETURN;
					END_IF
				END_FOR

			2: // Close iomap and arcfg
				Internal.AR_CloseArCfg_Int.Enable := TRUE;
				Internal.AR_CloseArCfg_Int.Ident := Internal.ArCfgIdent;
				Internal.AR_CloseArCfg_Int.Store := FALSE;
				Internal.IO_CloseIoMap_Int.Enable := TRUE;
				Internal.IO_CloseIoMap_Int.Ident := Internal.IoMapIdent;
				Internal.IO_CloseIoMap_Int.Store := FALSE;

				Internal.AR_CloseArCfg_Int();
				Internal.IO_CloseIoMap_Int();

				IF (Internal.AR_CloseArCfg_Int.Status = ERR_OK) AND (Internal.IO_CloseIoMap_Int.Status = ERR_OK) THEN
					Ready := TRUE;
					Initializing := FALSE;
					Internal.IoMapIdent := 0;
					Internal.ArCfgIdent := 0;
				END_IF
		END_CASE;
	ELSE // Ready = TRUE
		// Check if current indices are populated
		WHILE (brsstrlen(ADR(IoModules[Internal.IdxModule].IoChannels[Internal.IdxIoChannel].ChannelName)) = 0)
			OR (SelectedRefreshMode AND NOT IoModules[Internal.IdxModule].IoChannels[Internal.IdxIoChannel].IoForcing.RefreshActualValue AND NOT (Internal.CommandState = 1)) DO
			Internal.IdxModule := Internal.IdxModule + 1;
			Internal.IdxIoChannel := 0;
			IF Internal.IdxModule > gatMAX_IDX_IO_MODULES THEN
				Internal.IdxModule := 0;
				RETURN;
			END_IF
		END_WHILE

		// Set force value
		IF IoModules[Internal.IdxModule].IoChannels[Internal.IdxIoChannel].IoForcing.ForceValue <> Internal.ForceValue[Internal.IdxModule, Internal.IdxIoChannel] THEN
			Internal.AsIOSetForceValue_Int.enable := TRUE;
			Internal.AsIOSetForceValue_Int.pDatapoint := ADR(IoModules[Internal.IdxModule].IoChannels[Internal.IdxIoChannel].IoForcing.DpName);
			Internal.AsIOSetForceValue_Int.value := IoModules[Internal.IdxModule].IoChannels[Internal.IdxIoChannel].IoForcing.ForceValue;
			Internal.AsIOSetForceValue_Int();
			IF Internal.AsIOSetForceValue_Int.status = ERR_OK THEN
				Internal.AsIOSetForceValue_Int.enable := FALSE;
				Internal.AsIOSetForceValue_Int();
				Internal.ForceValue[Internal.IdxModule, Internal.IdxIoChannel] := IoModules[Internal.IdxModule].IoChannels[Internal.IdxIoChannel].IoForcing.ForceValue;
			END_IF
		END_IF
		// Enable/Disable forcing
		IF IoModules[Internal.IdxModule].IoChannels[Internal.IdxIoChannel].IoForcing.SetForceActive <> Internal.ForceEnabled[Internal.IdxModule, Internal.IdxIoChannel] THEN
			IF IoModules[Internal.IdxModule].IoChannels[Internal.IdxIoChannel].IoForcing.SetForceActive THEN
				Internal.AsIOEnableForcing_Int.enable := TRUE;
				Internal.AsIOEnableForcing_Int.pDatapoint := ADR(IoModules[Internal.IdxModule].IoChannels[Internal.IdxIoChannel].IoForcing.DpName);
				Internal.AsIOEnableForcing_Int();
				IF (Internal.AsIOEnableForcing_Int.status = ERR_OK) THEN
					Internal.AsIOEnableForcing_Int.enable := FALSE;
					Internal.AsIOEnableForcing_Int();
					Internal.ForceEnabled[Internal.IdxModule, Internal.IdxIoChannel] := TRUE;
				END_IF
			ELSE
				Internal.AsIODisableForcing_Int.enable := TRUE;
				Internal.AsIODisableForcing_Int.pDatapoint := ADR(IoModules[Internal.IdxModule].IoChannels[Internal.IdxIoChannel].IoForcing.DpName);
				Internal.AsIODisableForcing_Int();
				IF (Internal.AsIODisableForcing_Int.status = ERR_OK) THEN
					Internal.AsIODisableForcing_Int.enable := FALSE;
					Internal.AsIODisableForcing_Int();
					Internal.ForceEnabled[Internal.IdxModule, Internal.IdxIoChannel] := FALSE;
				END_IF
			END_IF
		END_IF
		// Set actual value
		Internal.AsIODPStatus_Int.enable := TRUE;
		Internal.AsIODPStatus_Int.pDatapoint := ADR(IoModules[Internal.IdxModule].IoChannels[Internal.IdxIoChannel].IoForcing.DpName);
		Internal.AsIODPStatus_Int();
		IF Internal.AsIODPStatus_Int.status = ERR_OK THEN
			IF Internal.AsIODPStatus_Int.flags.2 THEN
				IoModules[Internal.IdxModule].IoChannels[Internal.IdxIoChannel].IoForcing.ActualValue := Internal.AsIODPStatus_Int.forceValue;
			ELSE
				IoModules[Internal.IdxModule].IoChannels[Internal.IdxIoChannel].IoForcing.ActualValue := Internal.AsIODPStatus_Int.value;
			END_IF
			Internal.AsIODPStatus_Int.enable := FALSE;
			Internal.AsIODPStatus_Int();
		END_IF
		// Go to next index when nothing to do
		IF ((Internal.AsIOSetForceValue_Int.status = ERR_FUB_ENABLE_FALSE) OR (Internal.AsIOSetForceValue_Int.status = ERR_OK))
			AND ((Internal.AsIOEnableForcing_Int.status = ERR_FUB_ENABLE_FALSE) OR (Internal.AsIOEnableForcing_Int.status = ERR_OK))
			AND ((Internal.AsIODisableForcing_Int.status = ERR_FUB_ENABLE_FALSE) OR (Internal.AsIODisableForcing_Int.status = ERR_OK))
			AND ((Internal.AsIODPStatus_Int.status = ERR_FUB_ENABLE_FALSE) OR (Internal.AsIODPStatus_Int.status = ERR_OK)) THEN
			Internal.IdxIoChannel := Internal.IdxIoChannel + 1;
			IF Internal.IdxIoChannel > gatMAX_IDX_IO_CHANNELS THEN
				Internal.IdxIoChannel := 0;
				Internal.IdxModule := Internal.IdxModule + 1;
			END_IF
			IF Internal.IdxModule > gatMAX_IDX_IO_MODULES THEN
				Internal.IdxModule := 0;
			END_IF
			// Handle command inputs
			CASE Internal.CommandState OF
				0: // Wait for command
					IF ResetAllForcing THEN
						FOR Internal.IdxModuleCmd := 0 TO gatMAX_IDX_IO_MODULES DO
							FOR Internal.IdxIoChannelCmd := 0 TO gatMAX_IDX_IO_CHANNELS DO
								IoModules[Internal.IdxModuleCmd].IoChannels[Internal.IdxIoChannelCmd].IoForcing.SetForceActive := FALSE;
							END_FOR
						END_FOR
						CommandBusy := TRUE;
						Internal.CommandState := 1;
					END_IF
				1: // ResetAllForcing
					CommandBusy := TRUE;
					FOR Internal.IdxModuleCmd := 0 TO gatMAX_IDX_IO_MODULES DO
						FOR Internal.IdxIoChannelCmd := 0 TO gatMAX_IDX_IO_CHANNELS DO
							IF Internal.ForceEnabled[Internal.IdxModuleCmd, Internal.IdxIoChannelCmd] THEN
								RETURN;
							END_IF
						END_FOR
					END_FOR
					// All forcing is disabled
					CommandBusy := FALSE;
					CommandDone := TRUE;
					Internal.CommandState := 10;
				10: // Command done
					CommandDone := TRUE;
					IF NOT ResetAllForcing THEN
						CommandDone := FALSE;
						Internal.CommandState := 0;
					END_IF
			END_CASE;
		END_IF
	END_IF
END_FUNCTION_BLOCK

// Creates the IO data point name from the given information
FUNCTION GatMakeIoDpName
	brsmemset(ADR(DpName), 0, SIZEOF(DpName));

	CASE IoChannel.Type OF
		IO_DIG_INPUT:
			brsstrcpy(ADR(DpName), ADR('%IX.'));

		IO_DIG_OUTPUT:
			brsstrcpy(ADR(DpName), ADR('%QX.'));

		IO_ANA_INPUT:
			brsstrcpy(ADR(DpName), ADR('%IW.'));

		IO_TEMP_INPUT:
			brsstrcpy(ADR(DpName), ADR('%IW.'));

		IO_RESISTOR_INPUT:
			brsstrcpy(ADR(DpName), ADR('%IW.'));

		IO_ANA_OUTPUT:
			brsstrcpy(ADR(DpName), ADR('%QW.'));

		IO_PWM_OUTPUT:
			brsstrcpy(ADR(DpName), ADR('%QW.'));

		IO_USINT_INPUT:
			brsstrcpy(ADR(DpName), ADR('%IB.'));

		IO_USINT_OUTPUT:
			brsstrcpy(ADR(DpName), ADR('%QB.'));

		IO_UDINT_INPUT:
			brsstrcpy(ADR(DpName), ADR('%ID.'));

		IO_UDINT_OUTPUT:
			brsstrcpy(ADR(DpName), ADR('%QD.'));
	END_CASE;

	brsstrcat(ADR(DpName), ADR(IoChannel.ModulePath));
	brsstrcat(ADR(DpName), ADR('.'));
	brsstrcat(ADR(DpName), ADR(IoChannel.ChannelName));

	GatMakeIoDpName := TRUE;
END_FUNCTION

// Determines whether an IO channel should be accessible on the HMI
FUNCTION GatIoIsVisible
	GatIoIsVisible := TRUE;
	IF (brsmemcmp(ADR(ChannelName), ADR('DigitalOutput'), 13) = 0) THEN
		RETURN;
	END_IF
	IF (brsmemcmp(ADR(ChannelName), ADR('DigitalInput'), 12) = 0) THEN
		RETURN;
	END_IF
	IF (brsmemcmp(ADR(ChannelName), ADR('CounterInput'), 12) = 0) THEN
		RETURN;
	END_IF
	IF (brsmemcmp(ADR(ChannelName), ADR('AnalogOutput'), 12) = 0) THEN
		RETURN;
	END_IF
	IF (brsmemcmp(ADR(ChannelName), ADR('AnalogInput'), 11) = 0) THEN
		RETURN;
	END_IF
	IF (brsmemcmp(ADR(ChannelName), ADR('Temperature'), 11) = 0) THEN
		RETURN;
	END_IF
	IF (brsmemcmp(ADR(ChannelName), ADR('RelayOutput'), 11) = 0) THEN
		RETURN;
	END_IF
	IF (brsmemcmp(ADR(ChannelName), ADR('PulseWidthCurrentPwm'), 20) = 0) THEN
		RETURN;
	END_IF
	IF (brsmemcmp(ADR(ChannelName), ADR('PulseWidthCurrentPWM'), 20) = 0) THEN
		RETURN;
	END_IF
	IF (brsmemcmp(ADR(ChannelName), ADR('Counter'), 7) = 0) THEN
		RETURN;
	END_IF
	GatIoIsVisible := FALSE;
	RETURN;
END_FUNCTION
```
